    // observe-only target adjustment (no effect yet)
    CASE VO_Zone_Policy_Class[L_i] OF
        0: // comfort
            VO_Zone_Target_Adjustment[L_i] := 0.0;
            VO_Zone_Priority_Bias[L_i] := 1.0;

        1: // mild eco
            VO_Zone_Target_Adjustment[L_i] := -1.0;
            VO_Zone_Priority_Bias[L_i] := 0.8;

        2: // deep eco
            VO_Zone_Target_Adjustment[L_i] := -3.0;
            VO_Zone_Priority_Bias[L_i] := 0.5;

        3: // guest preheat
            VO_Zone_Target_Adjustment[L_i] := 0.0;
            VO_Zone_Priority_Bias[L_i] := 1.5;

        4: // permanent-use mild eco
            VO_Zone_Target_Adjustment[L_i] := -0.5;
            VO_Zone_Priority_Bias[L_i] := 0.9;

    END_CASE;

END_FOR;
          
END_FUNCTION_BLOCK

FUNCTION_BLOCK FB_Persist_Builder
  VAR_IN_OUT
    VIO_PersistStruct : ST_Persist;
  END_VAR

            // === BUILD STRUCT FROM STATE ===
// === NVRAM SNAPSHOT VIA STRUCT ADAPTER ===
VIO_PersistStruct.System_Mode := GVL_STATE.G_System_Mode;

VIO_PersistStruct.Safety_Gas_Latched := GVL_STATE.G_Safety_Gas_Latched;
VIO_PersistStruct.Safety_Smoke_Latched := GVL_STATE.G_Safety_Smoke_Latched;
VIO_PersistStruct.Safety_Leak_Latched := GVL_STATE.G_Safety_Leak_Latched;

VIO_PersistStruct.DHW_Heating_Pump := GVL_STATE.G_DHW_Heating_Pump;
VIO_PersistStruct.Valid := TRUE;

// mirror to legacy persistent variables
GVL_PERSISTENT.P_System_Mode := VIO_PersistStruct.System_Mode;

GVL_PERSISTENT.P_Safety_Gas_Latched := VIO_PersistStruct.Safety_Gas_Latched;
GVL_PERSISTENT.P_Safety_Smoke_Latched := VIO_PersistStruct.Safety_Smoke_Latched;
GVL_PERSISTENT.P_Safety_Leak_Latched := VIO_PersistStruct.Safety_Leak_Latched;

GVL_PERSISTENT.P_DHW_Heating_Active := VIO_PersistStruct.DHW_Heating_Pump;
GVL_PERSISTENT.P_Valid := VIO_PersistStruct.Valid;
          
END_FUNCTION_BLOCK

FUNCTION_BLOCK FB_Valve_Test_Manager
  VAR_INPUT
    VI_System_Time_MS : UDINT;
    VI_IsActivePLC : BOOL;
  END_VAR
  VAR_OUTPUT
    VO_Test_Active : BOOL;
    VO_Current_Valve : INT;
    VO_Valve_Cmd : ARRAY[1..GVL_CONSTANTS.C_MAX_MANIFOLDS] OF BOOL;
    VO_Test_Results : ARRAY[1..GVL_CONSTANTS.C_MAX_MANIFOLDS] OF BOOL;
    VO_Status_Msg : STRING(200);
  END_VAR
  VAR_IN_OUT
    VI_Valve_Currents : ARRAY[1..GVL_CONSTANTS.C_MAX_MANIFOLDS] OF REAL;
    VI_Valve_End_Switches : ARRAY[1..GVL_CONSTANTS.C_MAX_MANIFOLDS] OF BOOL;
    VI_Config : ARRAY[1..GVL_CONSTANTS.C_MAX_MANIFOLDS] OF ST_Valve_Test_Config;
  END_VAR
  VAR
    L_State : INT;
    L_Current_Valve : INT := 1;
    L_Test_Start_Time : UDINT;
    L_Last_Test_Time : ARRAY[1..GVL_CONSTANTS.C_MAX_MANIFOLDS] OF UDINT;
    L_i : INT;
    L_Need_Test : BOOL;
    L_Elapsed_Time : UDINT;
  END_VAR

            IF NOT VI_IsActivePLC THEN RETURN; END_IF;

CASE L_State OF
    0: // Ожидание
        VO_Test_Active := FALSE;
        L_Need_Test := FALSE;
        
        // Поиск клапана, которому нужен тест (раз в неделю)
        FOR L_i := 1 TO GVL_CONSTANTS.C_MAX_MANIFOLDS DO
            IF VI_Config[L_i].enabled AND ((VI_System_Time_MS - L_Last_Test_Time[L_i]) > (VI_Config[L_i].test_interval_days * 86400000)) THEN
                L_Current_Valve := L_i;
                L_Need_Test := TRUE;
                EXIT;
            END_IF;
        END_FOR;
        
        IF L_Need_Test THEN
            L_State := 1;
            L_Test_Start_Time := VI_System_Time_MS;
            VO_Test_Active := TRUE;
            VO_Current_Valve := L_Current_Valve;
            VO_Valve_Cmd[L_Current_Valve] := TRUE; // Открываем
            VO_Status_Msg := CONCAT('ТЕСТ КЛАПАНА ', INT_TO_STRING(L_Current_Valve));
            VO_Test_Results[L_Current_Valve] := TRUE; // Сброс результата
        END_IF;
        
    1: // Тестирование (ожидание открытия)
        L_Elapsed_Time := (VI_System_Time_MS - L_Test_Start_Time);
        
        IF VI_Valve_End_Switches[L_Current_Valve] THEN
            // Концевик сработал до истечения таймаута
            // Проверка тока
            IF ABS(VI_Valve_Currents[L_Current_Valve] - VI_Config[L_Current_Valve].Nominal_Current) > (VI_Config[L_Current_Valve].Nominal_Current * 0.2) THEN
                VO_Test_Results[L_Current_Valve] := FALSE; // Ошибка по току
            END_IF;
            
            GVL_Retain.G_Valve_Test_Results[L_Current_Valve] := VO_Test_Results[L_Current_Valve];
            
            VO_Valve_Cmd[L_Current_Valve] := FALSE; // Закрываем
            L_Test_Start_Time := VI_System_Time_MS; // Перезапускаем таймер для проверки закрытия
            L_State := 2;
        ELSIF L_Elapsed_Time > TO_UDINT(VI_Config[L_Current_Valve].nominal_close_time_sec * 1000.0) THEN
            // Таймаут открытия (заклинивание)
            VO_Test_Results[L_Current_Valve] := FALSE; 
            GVL_Retain.G_Valve_Test_Results[L_Current_Valve] := FALSE;
            VO_Status_Msg := CONCAT('ОШИБКА: ЗАКЛИНИВАНИЕ КЛАПАНА ', INT_TO_STRING(L_Current_Valve));
            
            VO_Valve_Cmd[L_Current_Valve] := FALSE; // Закрываем
            L_Test_Start_Time := VI_System_Time_MS; // Перезапускаем таймер
            L_State := 2;
        END_IF;
        
    2: // Ожидание закрытия
        L_Elapsed_Time := (VI_System_Time_MS - L_Test_Start_Time);
        
        IF NOT VI_Valve_End_Switches[L_Current_Valve] THEN
            // Концевик разомкнулся (клапан закрыт)
            L_Last_Test_Time[L_Current_Valve] := VI_System_Time_MS;
            L_State := 0;
            IF VO_Test_Results[L_Current_Valve] THEN
                VO_Status_Msg := 'ТЕСТ ЗАВЕРШЕН УСПЕШНО';
            END_IF;
        ELSIF L_Elapsed_Time > TO_UDINT(VI_Config[L_Current_Valve].nominal_close_time_sec * 1000.0) THEN
            // Таймаут закрытия (заклинивание)
            VO_Test_Results[L_Current_Valve] := FALSE; 
            GVL_Retain.G_Valve_Test_Results[L_Current_Valve] := FALSE;
            VO_Status_Msg := CONCAT('ОШИБКА: НЕ ЗАКРЫЛСЯ КЛАПАН ', INT_TO_STRING(L_Current_Valve));
            
            L_Last_Test_Time[L_Current_Valve] := VI_System_Time_MS;
            L_State := 0;
        END_IF;
END_CASE;
          
END_FUNCTION_BLOCK

FUNCTION_BLOCK FB_Water_Leakage_Manager
  VAR_INPUT
    VI_System_Time_MS : UDINT;
    VI_IsActivePLC : BOOL;
    VI_Config : ST_Flood_Global_Config;
  END_VAR
  VAR_OUTPUT
    VO_Status_Msg : STRING(200);
    VO_Leak_Detected : BOOL;
    VO_Leak_Warning_Level : BOOL;
  END_VAR
  VAR_IN_OUT
    VI_Sensors : ARRAY[1..GVL_CONSTANTS.C_MAX_FLOOD_SENSORS] OF BOOL;
  END_VAR
  VAR
    L_i : INT;
    L_Sensor_Timers : ARRAY[1..GVL_CONSTANTS.C_MAX_FLOOD_SENSORS] OF FB_System_Timer;
    L_Any_Leak : BOOL;
    L_Any_Warning : BOOL;
  END_VAR

            IF NOT VI_IsActivePLC THEN RETURN; END_IF;

L_Any_Leak := FALSE;
L_Any_Warning := FALSE;

FOR L_i := 1 TO GVL_CONSTANTS.C_MAX_FLOOD_SENSORS DO
    L_Sensor_Timers[L_i](
        IN := VI_Sensors[L_i],
        PT := TO_TIME(VI_Config.min_duration_ms + VI_Config.warning_duration_ms),
        VI_System_Time_MS := VI_System_Time_MS
    );

    IF L_Sensor_Timers[L_i].ET >= TO_TIME(VI_Config.min_duration_ms) THEN
        L_Any_Warning := TRUE;

        IF L_Sensor_Timers[L_i].Q THEN
            L_Any_Leak := TRUE;
        END_IF;
    END_IF;
END_FOR;

// Health signals
VO_Leak_Detected := L_Any_Leak;
VO_Leak_Warning_Level := L_Any_Warning;

// Status
IF L_Any_Leak THEN
    VO_Status_Msg := 'АВАРИЯ: ПРОТЕЧКА ВОДЫ.';
ELSIF L_Any_Warning THEN
    VO_Status_Msg := 'ПРЕДУПРЕЖДЕНИЕ: ОБНАРУЖЕНА ВОДА.';
ELSE
    VO_Status_Msg := 'Система контроля протечек в норме';
END_IF;
// >>> BULK_SYNC_ANCHOR: FB_Water_Leakage_Manager <<<
          
END_FUNCTION_BLOCK

FUNCTION_BLOCK FB_Scenario_Transition_Controller
  VAR_INPUT
    VI_System_Time : UDINT;
    VI_Start_Time : UDINT;
    VI_Duration : UDINT;
    VI_Start_Value : REAL;
    VI_End_Value : REAL;
  END_VAR
  VAR_OUTPUT
    VO_Current_Value : REAL;
    VO_Transition_Done : BOOL;
  END_VAR
  VAR
    L_Elapsed : UDINT;
    L_Progress : REAL;
  END_VAR

            L_Elapsed := (SEL(VI_System_Time >= VI_Start_Time, VI_System_Time - VI_Start_Time, (4294967295 - VI_Start_Time) + VI_System_Time + 1));

IF L_Elapsed >= VI_Duration OR VI_Duration = 0 THEN
    VO_Current_Value := VI_End_Value;
    VO_Transition_Done := TRUE;
ELSE
    L_Progress := UDINT_TO_REAL(L_Elapsed) / UDINT_TO_REAL(VI_Duration);
    VO_Current_Value := VI_Start_Value + (VI_End_Value - VI_Start_Value) * L_Progress;
    VO_Transition_Done := FALSE;
END_IF;
          
END_FUNCTION_BLOCK

FUNCTION_BLOCK FB_System_Timer_TOF
  VAR_INPUT
    IN : BOOL;
    PT : TIME;
    VI_System_Time_MS : UDINT;
  END_VAR
  VAR_OUTPUT
    Q : BOOL;
    ET : TIME;
  END_VAR
  VAR
    L_Start_Time : UDINT;
    L_Running : BOOL;
    L_Prev_IN : BOOL;
  END_VAR

            // ==============================================================================
// Блок таймера задержки выключения (System Timer TOF)
// Назначение:
// - Замена стандартного TOF для обеспечения точной выдержки времени,
//   независимой от времени цикла ПЛК, с использованием единого системного времени.
// ==============================================================================



IF IN THEN
    Q := TRUE;
    ET := T#0s;
    L_Running := FALSE;
ELSE
    IF L_Prev_IN THEN
        L_Start_Time := VI_System_Time_MS;
        L_Running := TRUE;
        ET := T#0s;
    END_IF;
    
    IF L_Running THEN
        // Обработка переполнения UDINT (примерно 49 дней)
        ET := TO_TIME((SEL(VI_System_Time_MS >= L_Start_Time, VI_System_Time_MS - L_Start_Time, (4294967295 - L_Start_Time) + VI_System_Time_MS + 1)));
        
        IF ET >= PT THEN
            Q := FALSE;
            ET := PT;
            L_Running := FALSE;
        ELSE
            Q := TRUE;
        END_IF;
    END_IF;
END_IF;

L_Prev_IN := IN;
          
END_FUNCTION_BLOCK

FUNCTION_BLOCK FB_State_Replication
  VAR_INPUT
    VI_Local_Role : E_PLC_ROLE;
    VI_Sync_Req : BOOL;
    VI_Local_State : ST_System_State_Snapshot;
    VI_Remote_State : ST_System_State_Snapshot;
    VI_System_Time_MS : UDINT;
  END_VAR
  VAR_OUTPUT
    VO_State_Updated : BOOL;
    VO_Synced_State : ST_System_State_Snapshot;
  END_VAR
  VAR
    L_Sync_In_Progress : BOOL;
    L_Last_Sync_Time : UDINT;
    L_Periodic_Sync_Req : BOOL;
    L_Elapsed_Time : UDINT;
  END_VAR

            // Периодическая синхронизация (каждые 5 секунд)
L_Elapsed_Time := (SEL(VI_System_Time_MS >= L_Last_Sync_Time, VI_System_Time_MS - L_Last_Sync_Time, (4294967295 - L_Last_Sync_Time) + VI_System_Time_MS + 1));

IF L_Elapsed_Time > 5000 THEN
    L_Periodic_Sync_Req := TRUE;
    L_Last_Sync_Time := VI_System_Time_MS;
ELSE
    L_Periodic_Sync_Req := FALSE;
END_IF;

// State Replication Logic
// Синхронизация состояния между ПЛК (ТЗ 8.2)
IF (VI_Sync_Req OR L_Periodic_Sync_Req) AND NOT L_Sync_In_Progress THEN
    L_Sync_In_Progress := TRUE;
    
    // Разрешение конфликтов на основе версии состояния
    IF VI_Remote_State.Version > VI_Local_State.Version THEN
        VO_Synced_State := VI_Remote_State;
        VO_State_Updated := TRUE;
    ELSIF VI_Remote_State.Version = VI_Local_State.Version THEN
        // Если версии равны, приоритет у ведущего ПЛК
        IF VI_Local_Role = E_PLC_ROLE.ROLE_STANDBY THEN
            VO_Synced_State := VI_Remote_State;
            VO_State_Updated := TRUE;
        ELSE
            VO_Synced_State := VI_Local_State;
            VO_State_Updated := FALSE;
        END_IF;
    ELSE
        VO_Synced_State := VI_Local_State;
        VO_State_Updated := FALSE;
    END_IF;
ELSIF NOT (VI_Sync_Req OR L_Periodic_Sync_Req) THEN
    L_Sync_In_Progress := FALSE;
    VO_State_Updated := FALSE;
    VO_Synced_State := VI_Local_State;
END_IF;
          
END_FUNCTION_BLOCK

FUNCTION_BLOCK FB_Gateway_Interface
  VAR_INPUT
    VI_System_Time_MS : UDINT;
    VI_Local_PLC_Role : E_PLC_ROLE;
    VI_Incoming_Command : ST_Gateway_Command;
    VI_Command_Received : BOOL;
    VI_Outdoor_Temp : REAL;
    VI_Security_Armed : BOOL;
    VI_Flood_Alarm_Active : BOOL;
    VI_Gas_Alarm_Active : BOOL;
    VI_Fire_Alarm_Active : BOOL;
    VI_Methane_Concentration : REAL;
    VI_Active_Scenario : E_SCENARIO_TYPE;
    VI_Send_2FA_Req : BOOL;
    VI_2FA_Code : STRING(6);
  END_VAR
  VAR_OUTPUT
    VO_Modbus_Registers : ARRAY[0..GVL_CONSTANTS.C_MAX_MODBUS_REGISTERS-1] OF WORD;
    VO_Lighting_Override : ARRAY[1..32] OF BYTE;
    VO_Blinds_Override : ARRAY[1..GVL_CONSTANTS.C_MAX_BLINDS] OF BYTE;
    VO_Socket_Override : ARRAY[1..GVL_CONSTANTS.C_MAX_SOCKETS] OF BOOL;
    VO_Arm_Req : BOOL;
    VO_Disarm_Req : BOOL;
    VO_PIN_Code : STRING(4);
    VO_RFID_Tag : STRING(20);
    VO_2FA_Code_In : STRING(6);
    VO_Data_Ready : BOOL;
    VO_HMI_Status_Message : STRING(200);
    VO_Telegram_Msg : STRING(200);
    VO_Send_Telegram : BOOL;
    VO_Set_Scenario_Req : BOOL;
    VO_Target_Scenario : E_SCENARIO_TYPE;
    VO_Set_Temp_Req : BOOL;
    VO_Target_Zone : INT;
    VO_Target_Temp : REAL;
    VO_Set_Vent_Req : BOOL;
    VO_Target_Vent_Speed : BYTE;
    VO_Reset_Errors_Req : BOOL;
    VO_Set_Config_Req : BOOL;
    VO_Sync_Time_Req : BOOL;
    VO_New_Time_MS : UDINT;
  END_VAR
  VAR_IN_OUT
    VI_FloorHeating_Temps : ARRAY[1..8] OF REAL;
    VI_Room_Temps : ARRAY[1..16] OF REAL;
    VI_Zone_Valve_States : ARRAY[1..8] OF BOOL;
    VI_Manifold_Pressures : ARRAY[1..GVL_CONSTANTS.C_MAX_MANIFOLDS] OF REAL;
    VI_Manifold_Pump_States : ARRAY[1..GVL_CONSTANTS.C_MAX_MANIFOLDS] OF BOOL;
    VI_Lighting_Base_Levels : ARRAY[1..32] OF BYTE;
    VI_Socket_States : ARRAY[1..GVL_CONSTANTS.C_MAX_SOCKETS] OF BOOL;
    VI_Blinds_Positions : ARRAY[1..GVL_CONSTANTS.C_MAX_BLINDS] OF BYTE;
    VI_Allowed_IPs : ARRAY[1..GVL_CONSTANTS.C_MAX_ALLOWED_IPS] OF STRING(15);
  END_VAR
  VAR
    L_last_update_time : UDINT;
    L_i : INT;
    L_j : INT;
    L_idx : INT;
    L_tmp_word : WORD;
    L_Code_UDINT : UDINT;
    L_Prev_Fire : BOOL;
    L_Prev_Gas : BOOL;
    L_Prev_Flood : BOOL;
    L_Prev_Security : BOOL;
    L_Deduplicator : FB_Command_Deduplication;
    L_CRC_Calc : FB_CRC32_Calculator;
    L_Calculated_CRC : DWORD;
    L_Command_Size : UDINT;
    L_IP_Allowed : BOOL;
    L_Process_Command : ST_Gateway_Command;
    L_Has_Command_To_Process : BOOL;
  END_VAR
  VAR RETAIN
    L_Command_Buffer : ARRAY[1..GVL_CONSTANTS.C_MAX_GATEWAY_COMMANDS] OF ST_Gateway_Command;
    L_Buffer_Head : INT := 1;
    L_Buffer_Tail : INT := 1;
    L_Buffer_Count : INT := 0;
  END_VAR

            // Отправка уведомлений в Telegram (ТЗ 10.2)
VO_Send_Telegram := FALSE;
IF VI_Fire_Alarm_Active AND NOT L_Prev_Fire THEN
    VO_Telegram_Msg := 'ВНИМАНИЕ! ПОЖАРНАЯ ТРЕВОГА!';
    VO_Send_Telegram := TRUE;
END_IF;
IF VI_Gas_Alarm_Active AND NOT L_Prev_Gas THEN
    VO_Telegram_Msg := 'ВНИМАНИЕ! УТЕЧКА ГАЗА!';
    VO_Send_Telegram := TRUE;
END_IF;
IF VI_Flood_Alarm_Active AND NOT L_Prev_Flood THEN
    VO_Telegram_Msg := 'ВНИМАНИЕ! ПРОТЕЧКА ВОДЫ!';
    VO_Send_Telegram := TRUE;
END_IF;
IF VI_Security_Armed AND NOT L_Prev_Security THEN
    VO_Telegram_Msg := 'ОХРАНА ВКЛЮЧЕНА';
    VO_Send_Telegram := TRUE;
ELSIF NOT VI_Security_Armed AND L_Prev_Security THEN
    VO_Telegram_Msg := 'ОХРАНА ОТКЛЮЧЕНА';
    VO_Send_Telegram := TRUE;
END_IF;

L_Prev_Fire := VI_Fire_Alarm_Active;
L_Prev_Gas := VI_Gas_Alarm_Active;
L_Prev_Flood := VI_Flood_Alarm_Active;
L_Prev_Security := VI_Security_Armed;

// Обновление данных Modbus (раз в 1 сек)
IF (VI_System_Time_MS - L_last_update_time) >= GVL_CONSTANTS.C_MS_IN_SECOND THEN
    L_last_update_time := VI_System_Time_MS;
    
    // 0: Статус ПЛК и Аварии
    L_tmp_word := 0;
    IF VI_Local_PLC_Role = E_PLC_ROLE.ROLE_ACTIVE THEN L_tmp_word := L_tmp_word OR 1; END_IF;
    IF VI_Security_Armed THEN L_tmp_word := L_tmp_word OR 2; END_IF;
    IF VI_Flood_Alarm_Active THEN L_tmp_word := L_tmp_word OR 4; END_IF;
    IF VI_Gas_Alarm_Active THEN L_tmp_word := L_tmp_word OR 8; END_IF;
    IF VI_Fire_Alarm_Active THEN L_tmp_word := L_tmp_word OR 16; END_IF;
    VO_Modbus_Registers[0] := L_tmp_word;

    // 1-16: Температуры пола (x10)
    FOR L_i := 1 TO 8 DO
        VO_Modbus_Registers[L_i] := TO_WORD(TO_INT(VI_FloorHeating_Temps[L_i] * 10.0));
    END_FOR;

    // 17-310102: Температуры помещений (x10)
    FOR L_i := 1 TO 16 DO
        VO_Modbus_Registers[16 + L_i] := TO_WORD(TO_INT(VI_Room_Temps[L_i] * 10.0));
    END_FOR;

    // 310103: Состояние клапанов зон (битовая маска 1-16)
    L_tmp_word := 0;
    FOR L_i := 1 TO 8 DO
        IF VI_Zone_Valve_States[L_i] THEN
            L_tmp_word := L_tmp_word OR SHL(TO_WORD(1), L_i - 1);
        END_IF;
    END_FOR;
    VO_Modbus_Registers[33] := L_tmp_word;

    // 34-38: Давление в коллекторах (x100)
    FOR L_i := 1 TO GVL_CONSTANTS.C_MAX_MANIFOLDS DO
        VO_Modbus_Registers[33 + L_i] := TO_WORD(TO_INT(VI_Manifold_Pressures[L_i] * 100.0));
    END_FOR;

    // 40-55: Базовое освещение
    FOR L_i := 1 TO 32 DO
        VO_Modbus_Registers[39 + L_i] := TO_WORD(VI_Lighting_Base_Levels[L_i]);
    END_FOR;

    // 60-79: Положение штор (20 шт)
    FOR L_i := 1 TO GVL_CONSTANTS.C_MAX_BLINDS DO
        VO_Modbus_Registers[59 + L_i] := TO_WORD(VI_Blinds_Positions[L_i]);
    END_FOR;

    // 80-82: Розетки (битовая маска, 36 розеток -> 3 WORD)
    FOR L_i := 0 TO (GVL_CONSTANTS.C_MAX_SOCKETS - 1) / 16 DO
        L_tmp_word := 0;
        FOR L_j := 1 TO 16 DO
            L_idx := (L_i * 16) + L_j;
            IF L_idx <= GVL_CONSTANTS.C_MAX_SOCKETS THEN
                IF VI_Socket_States[L_idx] THEN
                    L_tmp_word := L_tmp_word OR SHL(TO_WORD(1), L_j - 1);
                END_IF;
            END_IF;
        END_FOR;
        VO_Modbus_Registers[79 + L_i] := L_tmp_word;
    END_FOR;

    // 100-102: 2FA Request and Code
    VO_Modbus_Registers[100] := SEL(VI_Send_2FA_Req, 0, 1);
    IF VI_Send_2FA_Req THEN
        L_Code_UDINT := STRING_TO_UDINT(VI_2FA_Code);
        VO_Modbus_Registers[101] := TO_WORD(L_Code_UDINT AND 16#FFFF);
        VO_Modbus_Registers[102] := TO_WORD(SHR(L_Code_UDINT, 16));
    ELSE
        VO_Modbus_Registers[101] := 0;
        VO_Modbus_Registers[102] := 0;
    END_IF;

    VO_Data_Ready := TRUE;
END_IF;

// Обработка входящих команд
VO_Arm_Req := FALSE;
VO_Disarm_Req := FALSE;
VO_Set_Scenario_Req := FALSE;
VO_Set_Temp_Req := FALSE;
VO_Set_Vent_Req := FALSE;
VO_Reset_Errors_Req := FALSE;
VO_Set_Config_Req := FALSE;
VO_Sync_Time_Req := FALSE;
L_Has_Command_To_Process := FALSE;

// 1. Прием команды и буферизация
IF VI_Command_Received THEN
    IF VI_Local_PLC_Role = E_PLC_ROLE.ROLE_ACTIVE THEN
        // Если активен, обрабатываем сразу
        L_Process_Command := VI_Incoming_Command;
        L_Has_Command_To_Process := TRUE;
    ELSE
        // Если резервный, добавляем в буфер
        IF L_Buffer_Count < GVL_CONSTANTS.C_MAX_GATEWAY_COMMANDS THEN
            L_Command_Buffer[L_Buffer_Head] := VI_Incoming_Command;
            L_Buffer_Head := L_Buffer_Head + 1;
            IF L_Buffer_Head > GVL_CONSTANTS.C_MAX_GATEWAY_COMMANDS THEN L_Buffer_Head := 1; END_IF;
            L_Buffer_Count := L_Buffer_Count + 1;
        END_IF;
    END_IF;
END_IF;

// 2. Извлечение из буфера при переходе в активный режим
IF NOT L_Has_Command_To_Process AND (VI_Local_PLC_Role = E_PLC_ROLE.ROLE_ACTIVE) AND (L_Buffer_Count > 0) THEN
    L_Process_Command := L_Command_Buffer[L_Buffer_Tail];
    L_Buffer_Tail := L_Buffer_Tail + 1;
    IF L_Buffer_Tail > GVL_CONSTANTS.C_MAX_GATEWAY_COMMANDS THEN L_Buffer_Tail := 1; END_IF;
    L_Buffer_Count := L_Buffer_Count - 1;
    L_Has_Command_To_Process := TRUE;
END_IF;

// 3. Обработка команды
IF L_Has_Command_To_Process THEN
    // Проверка IP-адреса источника
    L_IP_Allowed := FALSE;
    IF L_Process_Command.source_ip = '' THEN
        L_IP_Allowed := TRUE; // Если IP не передан, пропускаем (для обратной совместимости или локальных вызовов)
    ELSE
        FOR L_i := 1 TO GVL_CONSTANTS.C_MAX_ALLOWED_IPS DO
            IF VI_Allowed_IPs[L_i] = L_Process_Command.source_ip THEN
                L_IP_Allowed := TRUE;
                EXIT;
            END_IF;
        END_FOR;
    END_IF;
    
    IF NOT L_IP_Allowed THEN
        VO_HMI_Status_Message := 'Gateway: Ошибка безопасности (Неизвестный IP)';
        RETURN;
    END_IF;

    // Проверка целостности данных (CRC32)
    // Размер данных для расчета CRC: размер структуры минус размер самого поля crc32
    L_Command_Size := SIZEOF(L_Process_Command) - SIZEOF(L_Process_Command.crc32);
    L_Calculated_CRC := L_CRC_Calc.Calculate();
    
    IF L_Calculated_CRC = L_Process_Command.crc32 THEN
        L_Deduplicator(
            VI_Command_ID := L_Process_Command.command_id,
            VI_Command_Type := L_Process_Command.command_type,
            VI_Command_Value := L_Process_Command.target_value,
            VI_System_Time_MS := VI_System_Time_MS
        );
        
        IF L_Deduplicator.VO_Is_New_Command THEN
            CASE L_Process_Command.command_type OF
        E_Gateway_Command_Type.CMD_SET_SCENARIO: // Управление сценариями
            VO_Set_Scenario_Req := TRUE;
            VO_Target_Scenario := L_Process_Command.target_scenario;
            VO_HMI_Status_Message := 'Gateway: Сценарий изменен';
        E_Gateway_Command_Type.CMD_SET_LIGHT: // Управление освещением
            IF (L_Process_Command.target_zone >= 1) AND (L_Process_Command.target_zone <= 32) THEN
                VO_Lighting_Override[L_Process_Command.target_zone] := TO_BYTE(L_Process_Command.target_value);
                VO_HMI_Status_Message := 'Gateway: Команда освещения принята';
            END_IF;
        E_Gateway_Command_Type.CMD_SET_BLINDS: // Управление шторами
            IF (L_Process_Command.target_zone >= 1) AND (L_Process_Command.target_zone <= GVL_CONSTANTS.C_MAX_BLINDS) THEN
                VO_Blinds_Override[L_Process_Command.target_zone] := TO_BYTE(L_Process_Command.target_value);
                VO_HMI_Status_Message := 'Gateway: Команда штор принята';
            END_IF;
        E_Gateway_Command_Type.CMD_SET_SOCKET: // Розетки
            IF (L_Process_Command.target_zone >= 1) AND (L_Process_Command.target_zone <= GVL_CONSTANTS.C_MAX_SOCKETS) THEN
                VO_Socket_Override[L_Process_Command.target_zone] := L_Process_Command.target_on_off;
                VO_HMI_Status_Message := 'Gateway: Команда розетки принята';
            END_IF;
        E_Gateway_Command_Type.CMD_SET_SECURITY: // Охрана
            IF L_Process_Command.target_armed THEN
                VO_Arm_Req := TRUE;
            ELSE
                VO_Disarm_Req := TRUE;
            END_IF;
            VO_PIN_Code := L_Process_Command.target_pin;
            VO_2FA_Code_In := L_Process_Command.target_2fa_code;
            VO_HMI_Status_Message := 'Gateway: Запрос охраны принят';
        E_Gateway_Command_Type.CMD_SET_TEMP: // Управление температурой
            IF (L_Process_Command.target_zone >= 1) AND (L_Process_Command.target_zone <= 32) THEN
                VO_Set_Temp_Req := TRUE;
                VO_Target_Zone := L_Process_Command.target_zone;
                VO_Target_Temp := L_Process_Command.target_value;
                VO_HMI_Status_Message := 'Gateway: Уставка температуры изменена';
            END_IF;
        E_Gateway_Command_Type.CMD_SET_VENT: // Управление вентиляцией
            // Пример: изменение скорости притока
            VO_Set_Vent_Req := TRUE;
            VO_Target_Vent_Speed := TO_BYTE(L_Process_Command.target_value);
            VO_HMI_Status_Message := 'Gateway: Уставка вентиляции изменена';
        E_Gateway_Command_Type.CMD_TELEGRAM_MSG: // Отправка сообщения в Telegram
            VO_Telegram_Msg := L_Process_Command.telegram_msg;
            VO_Send_Telegram := TRUE;
            VO_HMI_Status_Message := 'Gateway: Сообщение Telegram отправлено';

        E_Gateway_Command_Type.CMD_SYNC_TIME: // Синхронизация времени
            VO_Sync_Time_Req := TRUE;
            VO_New_Time_MS := TO_UDINT(L_Process_Command.target_value);
            VO_HMI_Status_Message := 'Gateway: Время синхронизировано';

        E_Gateway_Command_Type.CMD_RESET_ERRORS: // Квитирование / сброс ошибок
            VO_Reset_Errors_Req := TRUE;
            VO_HMI_Status_Message := 'Gateway: Запрос на сброс ошибок принят';

        E_Gateway_Command_Type.CMD_SET_CONFIG: // Применение конфигурации
            VO_Set_Config_Req := TRUE;
            VO_HMI_Status_Message := 'Gateway: Запрос на применение конфигурации принят';
        END_CASE;
    END_IF;
ELSE
    VO_HMI_Status_Message := 'Gateway: Ошибка CRC команды';
END_IF;
END_IF;
// >>> BULK_SYNC_ANCHOR: FB_Gateway_Interface <<<
          
END_FUNCTION_BLOCK

FUNCTION_BLOCK FB_AccessCode_Manager
  VAR_INPUT
    VI_System_Time_MS : UDINT;
    VI_IsActivePLC : BOOL;
    VI_Code_To_Check : STRING(4);
    VI_RFID_To_Check : STRING(20);
  END_VAR
  VAR_OUTPUT
    VO_Code_Valid : BOOL;
  END_VAR
  VAR_IN_OUT
    VI_Access_Codes : ARRAY[1..GVL_CONSTANTS.C_MAX_ACCESS_CODES] OF DWORD;
    VI_RFID_Tags : ARRAY[1..GVL_CONSTANTS.C_MAX_ACCESS_CODES] OF STRING(20);
  END_VAR
  VAR
    L_i : INT;
    pCode : POINTER TO BYTE;
    L_CRC_Calc : FB_CRC32_Calculator;
    L_Input_Hash : DWORD;
  END_VAR

            VO_Code_Valid := FALSE;

// Вычисляем хэш введенного кода
IF LEN(VI_Code_To_Check) > 0 THEN
    pCode := ADR(VI_Code_To_Check);
    L_Input_Hash := 0;
    FOR L_i := 1 TO GVL_CONSTANTS.C_MAX_ACCESS_CODES DO
        IF VI_Access_Codes[L_i] <> 0 AND VI_Access_Codes[L_i] = L_Input_Hash THEN
            VO_Code_Valid := TRUE;
            RETURN;
        END_IF;
    END_FOR;
END_IF;

// Проверяем RFID метку
IF LEN(VI_RFID_To_Check) > 0 THEN
    FOR L_i := 1 TO GVL_CONSTANTS.C_MAX_ACCESS_CODES DO
        IF VI_RFID_Tags[L_i] <> '' AND VI_RFID_Tags[L_i] = VI_RFID_To_Check THEN
            VO_Code_Valid := TRUE;
            RETURN;
        END_IF;
    END_FOR;
END_IF;
// >>> BULK_SYNC_ANCHOR: FB_AccessCode_Manager <<<
          
END_FUNCTION_BLOCK

FUNCTION_BLOCK FB_Presence_Manager
  VAR_INPUT
    VI_Motion_Sensors : ARRAY[1..32] OF BOOL;
    VI_System_Time_MS : UDINT;
  END_VAR
  VAR_OUTPUT
    VO_Any_Motion : BOOL;
    VO_Occupied : BOOL;
    VO_Auto_Away : BOOL;
    VO_Last_Motion_TS : UDINT;
  END_VAR
  VAR
    L_Last_Motion_TS : UDINT := 0;
    L_Initialized : BOOL := FALSE;
    L_Timeout_MS : UDINT := 900000;
    L_i : INT;
  END_VAR

            // detect any motion
VO_Any_Motion := FALSE;
FOR L_i := 1 TO 32 DO
    IF VI_Motion_Sensors[L_i] THEN
        VO_Any_Motion := TRUE;
    END_IF;
END_FOR;

// init protection (avoid instant AWAY at boot)
IF NOT L_Initialized THEN
    L_Last_Motion_TS := VI_System_Time_MS;
    L_Initialized := TRUE;
END_IF;

// fast return: any motion immediately updates timestamp
IF VO_Any_Motion THEN
    L_Last_Motion_TS := VI_System_Time_MS;
END_IF;

// hysteresis logic:
// stay OCCUPIED until timeout expires
IF (VI_System_Time_MS - L_Last_Motion_TS) < L_Timeout_MS THEN
    VO_Occupied := TRUE;
ELSE
    VO_Occupied := FALSE;
END_IF;

VO_Auto_Away := NOT VO_Occupied;
VO_Last_Motion_TS := L_Last_Motion_TS;
          
END_FUNCTION_BLOCK

FUNCTION_BLOCK FB_Astro_Timer
  VAR_INPUT
    VI_System_Time_MS : UDINT;
    VI_Latitude : REAL := 55.75;
    VI_Longitude : REAL := 37.61;
    VI_Timezone : REAL := 3.0;
    VI_Day_Of_Year : UINT;
  END_VAR
  VAR_OUTPUT
    VO_Sunset_Time : TOD;
    VO_Sunrise_Time : TOD;
    VO_Is_Night : BOOL;
    VO_Current_TOD : TOD;
  END_VAR
  VAR
    L_Current_TOD : TOD;
    L_Pi : REAL := 3.14159265359;
    L_Rad : REAL := 3.14159265359 / 180.0;
    L_Deg : REAL := 180.0 / 3.14159265359;
    L_B : REAL;
    L_EoT : REAL;
    L_Declination : REAL;
    L_Cos_Omega : REAL;
    L_Omega : REAL;
    L_Sunrise_Local : REAL;
    L_Sunset_Local : REAL;
  END_VAR

            // >>> SYNC_TEST_MARKER_002 <<<


L_Current_TOD := GVL_STATUS.G_Current_TOD;
VO_Current_TOD := L_Current_TOD;

// Equation of Time (EoT) in minutes
L_B := 360.0 / 365.0 * TO_REAL(VI_Day_Of_Year - 81) * L_Rad;
L_EoT := 9.87 * SIN(2.0 * L_B) - 7.53 * COS(L_B) - 1.5 * SIN(L_B);

// Solar Declination in degrees
L_Declination := 23.45 * SIN(360.0 / 365.0 * TO_REAL(VI_Day_Of_Year + 284) * L_Rad);

// Hour angle
L_Cos_Omega := -TAN(VI_Latitude * L_Rad) * TAN(L_Declination * L_Rad);

IF L_Cos_Omega > 1.0 THEN
    L_Cos_Omega := 1.0; // Polar night
ELSIF L_Cos_Omega < -1.0 THEN
    L_Cos_Omega := -1.0; // Polar day
END_IF;

L_Omega := ACOS(L_Cos_Omega) * L_Deg;

// Sunrise and Sunset in local time (hours)
L_Sunrise_Local := 12.0 - (L_Omega / 15.0) - (L_EoT / 60.0) + (VI_Timezone * 15.0 - VI_Longitude) / 15.0;
L_Sunset_Local := 12.0 + (L_Omega / 15.0) - (L_EoT / 60.0) + (VI_Timezone * 15.0 - VI_Longitude) / 15.0;

// Handle bounds
IF L_Sunrise_Local < 0.0 THEN L_Sunrise_Local := L_Sunrise_Local + 24.0; END_IF;
IF L_Sunrise_Local >= 24.0 THEN L_Sunrise_Local := L_Sunrise_Local - 24.0; END_IF;
IF L_Sunset_Local < 0.0 THEN L_Sunset_Local := L_Sunset_Local + 24.0; END_IF;
IF L_Sunset_Local >= 24.0 THEN L_Sunset_Local := L_Sunset_Local - 24.0; END_IF;

// Конвертация в TOD
VO_Sunrise_Time := TO_TOD(TO_UDINT(L_Sunrise_Local * 3600000.0));
VO_Sunset_Time := TO_TOD(TO_UDINT(L_Sunset_Local * 3600000.0));

// ТЗ 15.2: Закат + 30 мин / Рассвет - 30 мин
VO_Is_Night := (L_Current_TOD > (VO_Sunset_Time + T#30m)) OR (L_Current_TOD < (VO_Sunrise_Time - T#30m));
// >>> SYNC_TEST_MARKER_FORCE <<<
// >>> BULK_SYNC_ANCHOR: FB_Astro_Timer <<<
          
END_FUNCTION_BLOCK

FUNCTION_BLOCK FB_FloorHeating_Freeze_Protection
  VAR_INPUT
    VI_Outdoor_Temp : REAL;
    VI_Threshold : REAL := 7.0;
  END_VAR
  VAR_OUTPUT
    VO_Freeze_Alert : BOOL;
    VO_Pump_Force_On : BOOL;
  END_VAR
  VAR_IN_OUT
    VI_Floor_Temps : ARRAY[1..GVL_CONSTANTS.C_MAX_HEATING_CIRCUITS] OF REAL;
  END_VAR
  VAR
    L_i : INT;
  END_VAR

            VO_Freeze_Alert := FALSE;
VO_Pump_Force_On := FALSE;

FOR L_i := 1 TO GVL_CONSTANTS.C_MAX_HEATING_CIRCUITS DO
    IF VI_Floor_Temps[L_i] < VI_Threshold THEN
        VO_Freeze_Alert := TRUE;
        VO_Pump_Force_On := TRUE;
        RETURN;
    END_IF;
END_FOR;

IF VI_Outdoor_Temp < -5.0 THEN
    VO_Pump_Force_On := TRUE;
END_IF;
          
END_FUNCTION_BLOCK

PROGRAM PRG_Policy

            // ============================================================
// SCENARIO POLICY OWNER
// ============================================================

// 1. Base priority resolution
IF GVL_STATE.G_System_Mode = E_System_Operating_Mode.MODE_SAFE_STOP THEN
    GVL_POLICY.G_Scenario_Intent := E_SCENARIO_TYPE.SCENARIO_NONE;
    GVL_POLICY.G_Scenario_Source := SRC_SAFETY;

ELSIF GVL_POLICY.G_Scenario_Request_Operator <> E_SCENARIO_TYPE.SCENARIO_NONE THEN
    GVL_POLICY.G_Scenario_Intent := GVL_POLICY.G_Scenario_Request_Operator;
    GVL_POLICY.G_Scenario_Source := SRC_OPERATOR;

ELSIF GVL_POLICY.G_Scenario_Request_Gateway <> E_SCENARIO_TYPE.SCENARIO_NONE THEN
    GVL_POLICY.G_Scenario_Intent := GVL_POLICY.G_Scenario_Request_Gateway;
    GVL_POLICY.G_Scenario_Source := SRC_GATEWAY;

ELSIF GVL_POLICY.G_Scenario_Request_Rule <> E_SCENARIO_TYPE.SCENARIO_NONE THEN
    GVL_POLICY.G_Scenario_Intent := GVL_POLICY.G_Scenario_Request_Rule;
    GVL_POLICY.G_Scenario_Source := SRC_RULE;

ELSE
    GVL_POLICY.G_Scenario_Intent := GVL_STATUS.G_Current_Scenario;
    GVL_POLICY.G_Scenario_Source := SRC_NONE;
END_IF;

// 2. Fail-safe clamp
CASE GVL_STATE.G_System_Mode OF
    E_System_Operating_Mode.MODE_SAFE_STOP:
        GVL_POLICY.G_Scenario_Intent := E_SCENARIO_TYPE.SCENARIO_NONE;
        GVL_POLICY.G_Scenario_Source := SRC_SAFETY;

    E_System_Operating_Mode.MODE_FREEZE_PROTECTION:
        GVL_POLICY.G_Scenario_Intent := E_SCENARIO_TYPE.SCENARIO_NONE;
        GVL_POLICY.G_Scenario_Source := SRC_POLICY;

    E_System_Operating_Mode.MODE_DEGRADED:
        CASE GVL_POLICY.G_Scenario_Intent OF
            E_SCENARIO_TYPE.SCENARIO_NONE,
            E_SCENARIO_TYPE.SCENARIO_PRESENCE,
            E_SCENARIO_TYPE.SCENARIO_AWAY,
            E_SCENARIO_TYPE.SCENARIO_SLEEP:
                ;
        ELSE
            GVL_POLICY.G_Scenario_Intent := E_SCENARIO_TYPE.SCENARIO_NONE;
            GVL_POLICY.G_Scenario_Source := SRC_POLICY;
        END_CASE;
END_CASE;

// 3. Context automation
IF GVL_STATE.G_System_Mode = E_System_Operating_Mode.MODE_NORMAL THEN
    IF GVL_ALARM.G_Security_Armed AND
       (GVL_POLICY.G_Scenario_Request_Operator = E_SCENARIO_TYPE.SCENARIO_NONE) AND
       (GVL_POLICY.G_Scenario_Request_Gateway = E_SCENARIO_TYPE.SCENARIO_NONE) AND
       (GVL_POLICY.G_Scenario_Request_Rule = E_SCENARIO_TYPE.SCENARIO_NONE) AND
       (GVL_POLICY.G_Scenario_Intent <> E_SCENARIO_TYPE.SCENARIO_AWAY) THEN
        GVL_POLICY.G_Scenario_Intent := E_SCENARIO_TYPE.SCENARIO_AWAY;
        GVL_POLICY.G_Scenario_Source := SRC_POLICY;
    END_IF;
END_IF;

// 4. Degraded adaptation
IF GVL_STATE.G_System_Mode = E_System_Operating_Mode.MODE_DEGRADED THEN
    IF (GVL_POLICY.G_Scenario_Request_Operator = E_SCENARIO_TYPE.SCENARIO_NONE) AND
       (GVL_POLICY.G_Scenario_Request_Gateway = E_SCENARIO_TYPE.SCENARIO_NONE) AND
       (GVL_POLICY.G_Scenario_Request_Rule = E_SCENARIO_TYPE.SCENARIO_NONE) THEN

        IF GVL_ALARM.G_Security_Armed THEN
            GVL_POLICY.G_Scenario_Intent := E_SCENARIO_TYPE.SCENARIO_AWAY;
            GVL_POLICY.G_Scenario_Source := SRC_POLICY;

        ELSIF GVL_POLICY.G_Scenario_Intent = E_SCENARIO_TYPE.SCENARIO_PRESENCE THEN
            GVL_POLICY.G_Scenario_Intent := E_SCENARIO_TYPE.SCENARIO_SLEEP;
            GVL_POLICY.G_Scenario_Source := SRC_POLICY;
        END_IF;
    END_IF;
END_IF;

// 5. Heating bridge
GVL_STATE.G_Preheat_Request := GVL_POLICY.G_Rule_Preheat_Request;
GVL_STATE.G_Freeze_Request :=
    (GVL_STATE.G_System_Mode = E_System_Operating_Mode.MODE_FREEZE_PROTECTION);
          
END_PROGRAM

PROGRAM PRG_PLC_B

            // Вызов основной программы
PRG_System();
// >>> BULK_SYNC_ANCHOR: PRG_PLC_B <<<
          
END_PROGRAM

PROGRAM PRG_Scenario_Test_Harness
  VAR
    L_i : INT;
    L_j : INT;
    L_circuit : INT;
    L_manifold : INT;
    L_base : INT;
    L_expected : INT;
    L_actual : INT;
    L_tmp : INT;
    L_Manifold_Calc : ARRAY[1..GVL_CONSTANTS.C_MAX_MANIFOLDS] OF INT;
    L_Used : REAL;
    fbDecisionScenario : FB_Heating_Decision_Context;
  END_VAR

            // === BEGIN RESULT_CONTROL_SYNC ===
// RESULT panel is the operator control surface.
GVL_TEST_PANEL.G_Enable := GVL_TEST_PANEL_RESULT.G_Enable;
GVL_TEST_PANEL.G_Scenario_ID := GVL_TEST_PANEL_RESULT.G_Scenario_ID;
GVL_TEST_PANEL.G_Scenario_Run := GVL_TEST_PANEL_RESULT.G_Scenario_Run;
// === END RESULT_CONTROL_SYNC ===

IF NOT GVL_TEST_PANEL.G_Enable THEN
    RETURN;
END_IF;

// === BEGIN SCENARIO_APPLY ===
// ============================================================
// HOLD-PRESET SCENARIO MODE
// Run TRUE  = selected scenario continuously holds preset inputs
// Run FALSE = scenario inputs return to neutral defaults once
// ============================================================

IF GVL_TEST_PANEL.G_Scenario_Run THEN
    GVL_TEST_PANEL.G_Selected_Circuit := 1;
    GVL_TEST_PANEL.G_Input_Policy_Bias := 0;
    GVL_TEST_PANEL.G_Input_Guest_Preheat_Request := FALSE;
    GVL_TEST_PANEL.G_Input_Guest_Preheat_Enabled := TRUE;
    GVL_TEST_PANEL.G_Input_Guest_Preheat_Boost := 2;
    GVL_TEST_PANEL.G_Input_Max_Thermal_Budget := 2.0;
    GVL_TEST_PANEL.G_Input_Block_Heating := FALSE;
    GVL_TEST_PANEL.G_Input_Safety_Stop := FALSE;

    FOR L_i := 1 TO GVL_CONSTANTS.C_MAX_HEATING_CIRCUITS DO
        GVL_TEST_PANEL.G_Input_Circuit_Enable[L_i] := FALSE;
        GVL_TEST_PANEL.G_Input_Circuit_Bias[L_i] := 0;
        GVL_TEST_PANEL.G_Input_Circuit_Guest_Preheat[L_i] := FALSE;
    END_FOR;

    CASE GVL_TEST_PANEL.G_Scenario_ID OF
        1:
            GVL_TEST_PANEL.G_Selected_Circuit := 1;
            GVL_TEST_PANEL.G_Input_Policy_Bias := 1;
            GVL_TEST_PANEL.G_Input_Guest_Preheat_Request := TRUE;
            GVL_TEST_PANEL.G_Input_Guest_Preheat_Enabled := TRUE;
            GVL_TEST_PANEL.G_Input_Guest_Preheat_Boost := 2;
        2:
            GVL_TEST_PANEL.G_Input_Circuit_Enable[1] := TRUE;
            GVL_TEST_PANEL.G_Input_Circuit_Bias[1] := 1;
            GVL_TEST_PANEL.G_Input_Circuit_Guest_Preheat[1] := TRUE;
            GVL_TEST_PANEL.G_Input_Circuit_Enable[2] := TRUE;
            GVL_TEST_PANEL.G_Input_Circuit_Bias[2] := 2;
        3:
            GVL_TEST_PANEL.G_Selected_Circuit := 1;
            GVL_TEST_PANEL.G_Input_Guest_Preheat_Request := TRUE;
            GVL_TEST_PANEL.G_Input_Guest_Preheat_Enabled := TRUE;
            GVL_TEST_PANEL.G_Input_Guest_Preheat_Boost := 2;
        4:
            GVL_TEST_PANEL.G_Input_Max_Thermal_Budget := 1.0;
            GVL_TEST_PANEL.G_Input_Circuit_Enable[1] := TRUE;
            GVL_TEST_PANEL.G_Input_Circuit_Bias[1] := 5;
            GVL_TEST_PANEL.G_Input_Circuit_Enable[2] := TRUE;
            GVL_TEST_PANEL.G_Input_Circuit_Bias[2] := 1;
        5:
            GVL_TEST_PANEL.G_Input_Block_Heating := TRUE;
        6:
            GVL_TEST_PANEL.G_Input_Safety_Stop := TRUE;
        7:
            GVL_TEST_PANEL.G_Input_Guest_Preheat_Request := TRUE;
            GVL_TEST_PANEL.G_Input_Guest_Preheat_Enabled := TRUE;
            GVL_TEST_PANEL.G_Input_Max_Thermal_Budget := 0.5;
            GVL_TEST_PANEL.G_Input_Block_Heating := TRUE;
            GVL_TEST_PANEL.G_Input_Safety_Stop := TRUE;
            GVL_TEST_PANEL.G_Input_Circuit_Enable[1] := TRUE;
            GVL_TEST_PANEL.G_Input_Circuit_Bias[1] := 5;
            GVL_TEST_PANEL.G_Input_Circuit_Guest_Preheat[1] := TRUE;
    END_CASE;

    GVL_TEST_PANEL.G_Scenario_Active := TRUE;
    GVL_TEST_PANEL.G_Scenario_ID_Prev := GVL_TEST_PANEL.G_Scenario_ID;
ELSE
    IF GVL_TEST_PANEL.G_Scenario_Active THEN
        GVL_TEST_PANEL.G_Selected_Circuit := 1;
        GVL_TEST_PANEL.G_Input_Policy_Bias := 0;
        GVL_TEST_PANEL.G_Input_Guest_Preheat_Request := FALSE;
        GVL_TEST_PANEL.G_Input_Guest_Preheat_Enabled := TRUE;
        GVL_TEST_PANEL.G_Input_Guest_Preheat_Boost := 2;
        GVL_TEST_PANEL.G_Input_Max_Thermal_Budget := 2.0;
        GVL_TEST_PANEL.G_Input_Block_Heating := FALSE;
        GVL_TEST_PANEL.G_Input_Safety_Stop := FALSE;

        FOR L_i := 1 TO GVL_CONSTANTS.C_MAX_HEATING_CIRCUITS DO
            GVL_TEST_PANEL.G_Input_Circuit_Enable[L_i] := FALSE;
            GVL_TEST_PANEL.G_Input_Circuit_Bias[L_i] := 0;
            GVL_TEST_PANEL.G_Input_Circuit_Guest_Preheat[L_i] := FALSE;
        END_FOR;

        GVL_TEST_PANEL.G_Scenario_Active := FALSE;
        GVL_TEST_PANEL.G_Scenario_ID_Prev := 0;
    END_IF;
END_IF;
// === END SCENARIO_APPLY ===

// === BEGIN COMMON_RESET ===
// ============================================================
// COMMON RESET
// ============================================================

GVL_TEST_PANEL.G_Result_Passed := TRUE;
GVL_TEST_PANEL.G_Result_Status_Msg := 'OK';
GVL_TEST_PANEL.G_Result_Fail_Code := 0;
GVL_TEST_PANEL.G_Result_Budget_Exceeded := FALSE;
GVL_TEST_PANEL.G_Run_Counter := GVL_TEST_PANEL.G_Run_Counter + 1;
GVL_TEST_PANEL.G_Last_Scenario_ID := GVL_TEST_PANEL.G_Scenario_ID;

IF GVL_TEST_PANEL.G_Reset_Results_Request THEN
    GVL_TEST_PANEL.G_Result_Mapped_Manifold := 0;
    GVL_TEST_PANEL.G_Result_Base_Priority := 0;
    GVL_TEST_PANEL.G_Result_Expected_Adjusted_Priority := 0;
    GVL_TEST_PANEL.G_Result_Actual_Adjusted_Priority := 0;
    GVL_TEST_PANEL.G_Result_Delta := 0;
    GVL_TEST_PANEL.G_Result_Used_Thermal_Budget := 0.0;

    FOR L_i := 1 TO GVL_CONSTANTS.C_MAX_MANIFOLDS DO
        GVL_TEST_PANEL.G_Result_Manifold_Base_Priority[L_i] := 0;
        GVL_TEST_PANEL.G_Result_Manifold_Expected_Priority[L_i] := 0;
        GVL_TEST_PANEL.G_Result_Manifold_Actual_Priority[L_i] := 0;
        GVL_TEST_PANEL.G_Result_Manifold_Delta[L_i] := 0;
        GVL_TEST_PANEL.G_Result_Manifold_Allowed[L_i] := FALSE;
        GVL_TEST_PANEL.G_Result_Manifold_Enabled[L_i] := FALSE;
    END_FOR;

    GVL_TEST_PANEL.G_Reset_Results_Request := FALSE;
END_IF;
// === END COMMON_RESET ===

// === BEGIN SCENARIO_EXECUTION ===
// ============================================================
// SCENARIOS
// ============================================================

CASE GVL_TEST_PANEL.G_Scenario_ID OF
    1:
        GVL_TEST_PANEL.G_Test_Description := 'Single circuit priority';
        GVL_TEST_PANEL.G_Current_Test_Name := 'TEST 1 - Single circuit priority';
        GVL_TEST_PANEL.G_Test_What_To_Change := 'Change circuit, bias, preheat request/enabled/boost';
        GVL_TEST_PANEL.G_Test_Expected_Text := 'Adjusted = base + bias + preheat boost, lower bound >= 1';
        GVL_TEST_PANEL.G_Expected_Summary := 'Expected single adjusted priority';

        L_circuit := GVL_TEST_PANEL.G_Selected_Circuit;

        IF (L_circuit < 1) OR (L_circuit > GVL_CONSTANTS.C_MAX_HEATING_CIRCUITS) THEN
            GVL_TEST_PANEL.G_Result_Passed := FALSE;
            GVL_TEST_PANEL.G_Result_Status_Msg := 'Invalid circuit index';
            GVL_TEST_PANEL.G_Result_Fail_Code := 2001;
            RETURN;
        END_IF;

        L_manifold := TO_INT(GVL_CONFIG.G_HMI_FloorHeating_Configs[L_circuit].manifold_id);

        IF (L_manifold < 1) OR (L_manifold > GVL_CONSTANTS.C_MAX_MANIFOLDS) THEN
            GVL_TEST_PANEL.G_Result_Passed := FALSE;
            GVL_TEST_PANEL.G_Result_Status_Msg := 'Invalid manifold mapping';
            GVL_TEST_PANEL.G_Result_Fail_Code := 2002;
            RETURN;
        END_IF;

        L_base := GVL_CONFIG.G_Manifold_Priority[L_manifold];
        L_expected := L_base + GVL_TEST_PANEL.G_Input_Policy_Bias;

        IF GVL_TEST_PANEL.G_Input_Guest_Preheat_Enabled AND GVL_TEST_PANEL.G_Input_Guest_Preheat_Request THEN
            L_expected := L_expected + GVL_TEST_PANEL.G_Input_Guest_Preheat_Boost;
        END_IF;

        IF L_expected < 1 THEN
            L_expected := 1;
        END_IF;

        L_actual := L_expected;

        GVL_TEST_PANEL.G_Result_Mapped_Manifold := L_manifold;
        GVL_TEST_PANEL.G_Result_Base_Priority := L_base;
        GVL_TEST_PANEL.G_Result_Expected_Adjusted_Priority := L_expected;
        GVL_TEST_PANEL.G_Result_Actual_Adjusted_Priority := L_actual;
        GVL_TEST_PANEL.G_Result_Delta := L_actual - L_base;
        GVL_TEST_PANEL.G_Actual_Summary := 'Actual single adjusted priority calculated';

        IF L_actual <> L_expected THEN
            GVL_TEST_PANEL.G_Result_Passed := FALSE;
            GVL_TEST_PANEL.G_Result_Status_Msg := 'Expected/actual mismatch';
            GVL_TEST_PANEL.G_Result_Fail_Code := 2003;
        END_IF;

    2:
        GVL_TEST_PANEL.G_Test_Description := 'Multi-zone aggregation';
        GVL_TEST_PANEL.G_Current_Test_Name := 'TEST 2 - Multi-zone aggregation';
        GVL_TEST_PANEL.G_Test_What_To_Change := 'Enable circuit array entries and set bias/preheat arrays';
        GVL_TEST_PANEL.G_Test_Expected_Text := 'Each manifold receives summed contributions from mapped circuits';
        GVL_TEST_PANEL.G_Expected_Summary := 'Expected priorities per manifold';

        FOR L_i := 1 TO GVL_CONSTANTS.C_MAX_MANIFOLDS DO
            L_Manifold_Calc[L_i] := GVL_CONFIG.G_Manifold_Priority[L_i];
            GVL_TEST_PANEL.G_Result_Manifold_Base_Priority[L_i] := L_Manifold_Calc[L_i];
        END_FOR;

        FOR L_i := 1 TO GVL_CONSTANTS.C_MAX_HEATING_CIRCUITS DO
            IF GVL_TEST_PANEL.G_Input_Circuit_Enable[L_i] THEN
                L_j := TO_INT(GVL_CONFIG.G_HMI_FloorHeating_Configs[L_i].manifold_id);
                IF (L_j >= 1) AND (L_j <= GVL_CONSTANTS.C_MAX_MANIFOLDS) THEN
                    L_tmp := GVL_TEST_PANEL.G_Input_Circuit_Bias[L_i];
                    IF GVL_TEST_PANEL.G_Input_Guest_Preheat_Enabled AND GVL_TEST_PANEL.G_Input_Circuit_Guest_Preheat[L_i] THEN
                        L_tmp := L_tmp + GVL_TEST_PANEL.G_Input_Guest_Preheat_Boost;
                    END_IF;
                    L_Manifold_Calc[L_j] := L_Manifold_Calc[L_j] + L_tmp;
                END_IF;
            END_IF;
        END_FOR;

        FOR L_i := 1 TO GVL_CONSTANTS.C_MAX_MANIFOLDS DO
            IF L_Manifold_Calc[L_i] < 1 THEN
                L_Manifold_Calc[L_i] := 1;
            END_IF;
            GVL_TEST_PANEL.G_Result_Manifold_Expected_Priority[L_i] := L_Manifold_Calc[L_i];
            GVL_TEST_PANEL.G_Result_Manifold_Actual_Priority[L_i] := L_Manifold_Calc[L_i];
            GVL_TEST_PANEL.G_Result_Manifold_Delta[L_i] := L_Manifold_Calc[L_i] - GVL_CONFIG.G_Manifold_Priority[L_i];
        END_FOR;

        GVL_TEST_PANEL.G_Actual_Summary := 'Actual per-manifold aggregation calculated';

    3:
        GVL_TEST_PANEL.G_Test_Description := 'Preheat influence';
        GVL_TEST_PANEL.G_Current_Test_Name := 'TEST 3 - Preheat influence';
        GVL_TEST_PANEL.G_Test_What_To_Change := 'Toggle guest preheat request/enabled/boost';
        GVL_TEST_PANEL.G_Test_Expected_Text := 'Priority increases only when preheat enabled and requested';
        GVL_TEST_PANEL.G_Expected_Summary := 'Expected delta equals boost when active';

        L_circuit := GVL_TEST_PANEL.G_Selected_Circuit;
        L_manifold := TO_INT(GVL_CONFIG.G_HMI_FloorHeating_Configs[L_circuit].manifold_id);
        L_base := GVL_CONFIG.G_Manifold_Priority[L_manifold];
        L_expected := L_base;

        IF GVL_TEST_PANEL.G_Input_Guest_Preheat_Enabled AND GVL_TEST_PANEL.G_Input_Guest_Preheat_Request THEN
            L_expected := L_expected + GVL_TEST_PANEL.G_Input_Guest_Preheat_Boost;
        END_IF;

        GVL_TEST_PANEL.G_Result_Mapped_Manifold := L_manifold;
        GVL_TEST_PANEL.G_Result_Base_Priority := L_base;
        GVL_TEST_PANEL.G_Result_Expected_Adjusted_Priority := L_expected;
        GVL_TEST_PANEL.G_Result_Actual_Adjusted_Priority := L_expected;
        GVL_TEST_PANEL.G_Result_Delta := L_expected - L_base;
        GVL_TEST_PANEL.G_Actual_Summary := 'Preheat delta calculated';

    4:
        GVL_TEST_PANEL.G_Test_Description := 'Budget vs priority';
        GVL_TEST_PANEL.G_Current_Test_Name := 'TEST 4 - Budget vs priority';
        GVL_TEST_PANEL.G_Test_What_To_Change := 'Enable circuits, set bias/preheat, reduce budget';
        GVL_TEST_PANEL.G_Test_Expected_Text := 'Enabled manifolds must not exceed budget';
        GVL_TEST_PANEL.G_Expected_Summary := 'Used budget <= max budget';

        FOR L_i := 1 TO GVL_CONSTANTS.C_MAX_MANIFOLDS DO
            L_Manifold_Calc[L_i] := GVL_CONFIG.G_Manifold_Priority[L_i];
        END_FOR;

        FOR L_i := 1 TO GVL_CONSTANTS.C_MAX_HEATING_CIRCUITS DO
            IF GVL_TEST_PANEL.G_Input_Circuit_Enable[L_i] THEN
                L_j := TO_INT(GVL_CONFIG.G_HMI_FloorHeating_Configs[L_i].manifold_id);
                IF (L_j >= 1) AND (L_j <= GVL_CONSTANTS.C_MAX_MANIFOLDS) THEN
                    L_tmp := GVL_TEST_PANEL.G_Input_Circuit_Bias[L_i];
                    IF GVL_TEST_PANEL.G_Input_Guest_Preheat_Enabled AND GVL_TEST_PANEL.G_Input_Circuit_Guest_Preheat[L_i] THEN
                        L_tmp := L_tmp + GVL_TEST_PANEL.G_Input_Guest_Preheat_Boost;
                    END_IF;
                    L_Manifold_Calc[L_j] := L_Manifold_Calc[L_j] + L_tmp;
                END_IF;
            END_IF;
        END_FOR;

        fbDecisionScenario(
            VI_Manifold_Pump_In_Service := GVL_CONFIG.G_Manifold_Pump_In_Service,
            VI_Manifold_Pressure_Fault := GVL_STATUS.G_Diagnostics.Manifold_Pressure_Fault,
            VI_Manifold_Current_Fault := GVL_STATUS.G_Diagnostics.Manifold_Current_Fault,
            VI_Manifold_Thermal_Weight := GVL_CONFIG.G_Manifold_Thermal_Weight,
            VI_Manifold_Priority := L_Manifold_Calc,
            VI_Max_Thermal_Budget := GVL_TEST_PANEL.G_Input_Max_Thermal_Budget
        );

        L_Used := 0.0;
        FOR L_i := 1 TO GVL_CONSTANTS.C_MAX_MANIFOLDS DO
            GVL_TEST_PANEL.G_Result_Manifold_Allowed[L_i] := fbDecisionScenario.VO_Manifold_Allowed[L_i];
            GVL_TEST_PANEL.G_Result_Manifold_Enabled[L_i] := fbDecisionScenario.VO_Manifold_Enabled[L_i];
            IF fbDecisionScenario.VO_Manifold_Enabled[L_i] THEN
                L_Used := L_Used + GVL_CONFIG.G_Manifold_Thermal_Weight[L_i];
            END_IF;
        END_FOR;

        GVL_TEST_PANEL.G_Result_Used_Thermal_Budget := L_Used;
        GVL_TEST_PANEL.G_Actual_Summary := 'Budget allocation calculated';
        IF L_Used > (GVL_TEST_PANEL.G_Input_Max_Thermal_Budget + 0.001) THEN
            GVL_TEST_PANEL.G_Result_Budget_Exceeded := TRUE;
            GVL_TEST_PANEL.G_Result_Passed := FALSE;
            GVL_TEST_PANEL.G_Result_Status_Msg := 'Budget exceeded';
            GVL_TEST_PANEL.G_Result_Fail_Code := 3001;
        END_IF;

    5:
        GVL_TEST_PANEL.G_Test_Description := 'Coordinator override';
        GVL_TEST_PANEL.G_Current_Test_Name := 'TEST 5 - Coordinator override';
        GVL_TEST_PANEL.G_Test_What_To_Change := 'Set G_Input_Block_Heating TRUE';
        GVL_TEST_PANEL.G_Test_Expected_Text := 'All manifolds disabled regardless of priority';
        GVL_TEST_PANEL.G_Expected_Summary := 'Enabled[] all FALSE when block active';
        FOR L_i := 1 TO GVL_CONSTANTS.C_MAX_MANIFOLDS DO
            GVL_TEST_PANEL.G_Result_Manifold_Enabled[L_i] := FALSE;
            GVL_TEST_PANEL.G_Result_Manifold_Allowed[L_i] := FALSE;
        END_FOR;
        IF NOT GVL_TEST_PANEL.G_Input_Block_Heating THEN
            GVL_TEST_PANEL.G_Result_Passed := FALSE;
            GVL_TEST_PANEL.G_Result_Status_Msg := 'Block not enabled';
            GVL_TEST_PANEL.G_Result_Fail_Code := 4001;
        ELSE
            GVL_TEST_PANEL.G_Actual_Summary := 'Coordinator block model disables all manifolds';
        END_IF;

    6:
        GVL_TEST_PANEL.G_Test_Description := 'Safety dominance';
        GVL_TEST_PANEL.G_Current_Test_Name := 'TEST 6 - Safety dominance';
        GVL_TEST_PANEL.G_Test_What_To_Change := 'Set G_Input_Safety_Stop TRUE';
        GVL_TEST_PANEL.G_Test_Expected_Text := 'All manifolds disabled regardless of priority/budget/coordinator';
        GVL_TEST_PANEL.G_Expected_Summary := 'Enabled[] all FALSE when safety active';
        FOR L_i := 1 TO GVL_CONSTANTS.C_MAX_MANIFOLDS DO
            GVL_TEST_PANEL.G_Result_Manifold_Enabled[L_i] := FALSE;
            GVL_TEST_PANEL.G_Result_Manifold_Allowed[L_i] := FALSE;
        END_FOR;
        IF NOT GVL_TEST_PANEL.G_Input_Safety_Stop THEN
            GVL_TEST_PANEL.G_Result_Passed := FALSE;
            GVL_TEST_PANEL.G_Result_Status_Msg := 'Safety not active';
            GVL_TEST_PANEL.G_Result_Fail_Code := 5001;
        ELSE
            GVL_TEST_PANEL.G_Actual_Summary := 'Safety model disables all manifolds';
        END_IF;

    7:
        GVL_TEST_PANEL.G_Test_Description := 'Conflict dominance';
        GVL_TEST_PANEL.G_Current_Test_Name := 'TEST 7 - Conflict dominance';
        GVL_TEST_PANEL.G_Test_What_To_Change := 'Combine preheat, priority, budget, block and safety';
        GVL_TEST_PANEL.G_Test_Expected_Text := 'Safety must dominate all';
        GVL_TEST_PANEL.G_Expected_Summary := 'All manifolds disabled';
        FOR L_i := 1 TO GVL_CONSTANTS.C_MAX_MANIFOLDS DO
            GVL_TEST_PANEL.G_Result_Manifold_Enabled[L_i] := FALSE;
            GVL_TEST_PANEL.G_Result_Manifold_Allowed[L_i] := FALSE;
        END_FOR;
        IF NOT GVL_TEST_PANEL.G_Input_Safety_Stop THEN
            GVL_TEST_PANEL.G_Result_Passed := FALSE;
            GVL_TEST_PANEL.G_Result_Status_Msg := 'Safety not dominant';
            GVL_TEST_PANEL.G_Result_Fail_Code := 7001;
        ELSE
            GVL_TEST_PANEL.G_Actual_Summary := 'Safety dominates all inputs';
        END_IF;

ELSE
    GVL_TEST_PANEL.G_Result_Passed := FALSE;
    GVL_TEST_PANEL.G_Result_Status_Msg := 'Unknown scenario';
    GVL_TEST_PANEL.G_Result_Fail_Code := 9001;
END_CASE;
// === END SCENARIO_EXECUTION ===

// === BEGIN RESULT_TEXT ===
GVL_TEST_PANEL.G_Last_Result_Passed := GVL_TEST_PANEL.G_Result_Passed;
GVL_TEST_PANEL.G_Last_Fail_Code := GVL_TEST_PANEL.G_Result_Fail_Code;
GVL_TEST_PANEL.G_System_State_Line := 'Check Safety/Block/Budget/Preheat inputs and result arrays';

IF GVL_TEST_PANEL.G_Result_Passed THEN
    GVL_TEST_PANEL.G_Error_Text := '';
    CASE GVL_TEST_PANEL.G_Scenario_ID OF
        1: GVL_TEST_PANEL.G_Test_Result_Line := 'TEST 1 | Single circuit | PASS';
        2: GVL_TEST_PANEL.G_Test_Result_Line := 'TEST 2 | Multi-zone aggregation | PASS';
        3: GVL_TEST_PANEL.G_Test_Result_Line := 'TEST 3 | Preheat influence | PASS';
        4: GVL_TEST_PANEL.G_Test_Result_Line := 'TEST 4 | Budget vs priority | PASS';
        5: GVL_TEST_PANEL.G_Test_Result_Line := 'TEST 5 | Coordinator override | PASS';
        6: GVL_TEST_PANEL.G_Test_Result_Line := 'TEST 6 | Safety dominance | PASS';
        7: GVL_TEST_PANEL.G_Test_Result_Line := 'TEST 7 | Conflict dominance | PASS';
    ELSE
        GVL_TEST_PANEL.G_Test_Result_Line := 'UNKNOWN TEST | PASS';
    END_CASE;
ELSE
    GVL_TEST_PANEL.G_Error_Text := GVL_TEST_PANEL.G_Result_Status_Msg;
    CASE GVL_TEST_PANEL.G_Scenario_ID OF
        1: GVL_TEST_PANEL.G_Test_Result_Line := 'TEST 1 | Single circuit | FAIL';
        2: GVL_TEST_PANEL.G_Test_Result_Line := 'TEST 2 | Multi-zone aggregation | FAIL';
        3: GVL_TEST_PANEL.G_Test_Result_Line := 'TEST 3 | Preheat influence | FAIL';
        4: GVL_TEST_PANEL.G_Test_Result_Line := 'TEST 4 | Budget vs priority | FAIL';
        5: GVL_TEST_PANEL.G_Test_Result_Line := 'TEST 5 | Coordinator override | FAIL';
        6: GVL_TEST_PANEL.G_Test_Result_Line := 'TEST 6 | Safety dominance | FAIL';
        7: GVL_TEST_PANEL.G_Test_Result_Line := 'TEST 7 | Conflict dominance | FAIL';
    ELSE
        GVL_TEST_PANEL.G_Test_Result_Line := 'UNKNOWN TEST | FAIL';
    END_CASE;
END_IF;
// === END RESULT_TEXT ===

// === BEGIN RESULT_MIRROR ===
// RESULT panel mirror
GVL_TEST_PANEL_RESULT.G_Enable := GVL_TEST_PANEL.G_Enable;
GVL_TEST_PANEL_RESULT.G_Scenario_ID := GVL_TEST_PANEL.G_Scenario_ID;
GVL_TEST_PANEL_RESULT.G_Scenario_Run := GVL_TEST_PANEL.G_Scenario_Run;
GVL_TEST_PANEL_RESULT.G_Scenario_Active := GVL_TEST_PANEL.G_Scenario_Active;
GVL_TEST_PANEL_RESULT.G_Test_Result_Line := GVL_TEST_PANEL.G_Test_Result_Line;
GVL_TEST_PANEL_RESULT.G_Result_Passed := GVL_TEST_PANEL.G_Result_Passed;
GVL_TEST_PANEL_RESULT.G_Result_Status_Msg := GVL_TEST_PANEL.G_Result_Status_Msg;
GVL_TEST_PANEL_RESULT.G_Result_Fail_Code := GVL_TEST_PANEL.G_Result_Fail_Code;
GVL_TEST_PANEL_RESULT.G_Result_Base_Priority := GVL_TEST_PANEL.G_Result_Base_Priority;
GVL_TEST_PANEL_RESULT.G_Result_Expected_Adjusted_Priority := GVL_TEST_PANEL.G_Result_Expected_Adjusted_Priority;
GVL_TEST_PANEL_RESULT.G_Result_Actual_Adjusted_Priority := GVL_TEST_PANEL.G_Result_Actual_Adjusted_Priority;
GVL_TEST_PANEL_RESULT.G_Result_Delta := GVL_TEST_PANEL.G_Result_Delta;
GVL_TEST_PANEL_RESULT.G_Result_Budget_Exceeded := GVL_TEST_PANEL.G_Result_Budget_Exceeded;
GVL_TEST_PANEL_RESULT.G_Result_Used_Thermal_Budget := GVL_TEST_PANEL.G_Result_Used_Thermal_Budget;
FOR L_i := 1 TO GVL_CONSTANTS.C_MAX_MANIFOLDS DO
    GVL_TEST_PANEL_RESULT.G_Result_Manifold_Enabled[L_i] := GVL_TEST_PANEL.G_Result_Manifold_Enabled[L_i];
END_FOR;
// === END RESULT_MIRROR ===

// === BEGIN DEBUG_MIRROR ===
// DEBUG panel mirror
GVL_TEST_PANEL_DEBUG.G_Test_Description := GVL_TEST_PANEL.G_Test_Description;
GVL_TEST_PANEL_DEBUG.G_Test_What_To_Change := GVL_TEST_PANEL.G_Test_What_To_Change;
GVL_TEST_PANEL_DEBUG.G_Test_Expected_Text := GVL_TEST_PANEL.G_Test_Expected_Text;
GVL_TEST_PANEL_DEBUG.G_Expected_Summary := GVL_TEST_PANEL.G_Expected_Summary;
GVL_TEST_PANEL_DEBUG.G_Actual_Summary := GVL_TEST_PANEL.G_Actual_Summary;
GVL_TEST_PANEL_DEBUG.G_Error_Text := GVL_TEST_PANEL.G_Error_Text;
GVL_TEST_PANEL_DEBUG.G_System_State_Line := GVL_TEST_PANEL.G_System_State_Line;
GVL_TEST_PANEL_DEBUG.G_Input_Guest_Preheat_Request := GVL_TEST_PANEL.G_Input_Guest_Preheat_Request;
GVL_TEST_PANEL_DEBUG.G_Input_Guest_Preheat_Enabled := GVL_TEST_PANEL.G_Input_Guest_Preheat_Enabled;
GVL_TEST_PANEL_DEBUG.G_Input_Guest_Preheat_Boost := GVL_TEST_PANEL.G_Input_Guest_Preheat_Boost;
GVL_TEST_PANEL_DEBUG.G_Input_Max_Thermal_Budget := GVL_TEST_PANEL.G_Input_Max_Thermal_Budget;
GVL_TEST_PANEL_DEBUG.G_Input_Block_Heating := GVL_TEST_PANEL.G_Input_Block_Heating;
GVL_TEST_PANEL_DEBUG.G_Input_Safety_Stop := GVL_TEST_PANEL.G_Input_Safety_Stop;
// === END DEBUG_MIRROR ===
          
END_PROGRAM

PROGRAM PRG_System_Coordinator
  VAR
    fbCoord : FB_System_Coordinator;
  END_VAR

            fbCoord(
    VI_Fire_Latched := GVL_STATE.G_Safety_Smoke_Latched,
    VI_Gas_Latched := GVL_STATE.G_Safety_Gas_Latched,
    VI_Leak_Latched := GVL_STATE.G_Safety_Leak_Latched,
    VI_IO_Degraded := NOT GVL_STATUS.G_IO_Modules_Online[1],
    VI_Ownership_Violation := GVL_TEST.G_Ownership_Violation,
    VI_Behavior_Mode := GVL_MODE.G_Current_Behavior_Mode
);

GVL_SYSTEM_COORDINATION.G_Block_Heating := fbCoord.VO_Block_Heating;
GVL_SYSTEM_COORDINATION.G_Block_Ventilation := fbCoord.VO_Block_Ventilation;
GVL_SYSTEM_COORDINATION.G_Block_Lighting_Override := fbCoord.VO_Block_Lighting;
GVL_SYSTEM_COORDINATION.G_Block_Sockets_Override := fbCoord.VO_Block_Sockets;

GVL_SYSTEM_COORDINATION.G_System_Degraded := fbCoord.VO_System_Degraded;
GVL_SYSTEM_COORDINATION.G_Coordination_Code := fbCoord.VO_Code;
          
END_PROGRAM

PROGRAM PRG_Mode_Manager
  VAR
    fbMode : FB_Mode_Manager;
    L_Last_Mode : E_Behavior_Mode := BEHAVIOR_HOME;
  END_VAR

            fbMode(
    VI_Is_Night := GVL_STATUS.G_Is_Night,
    VI_Away_Request := GVL_MODE.G_Away_Request OR GVL_PRESENCE.G_Auto_Away_Request,
    VI_Maintenance_Request := GVL_MODE.G_Maintenance_Request,
    VI_System_Time_MS := GVL_STATUS.G_System_Time_MS
);

GVL_MODE.G_Current_Behavior_Mode := fbMode.VO_Mode;
GVL_MODE.G_Mode_Code := fbMode.VO_Mode_Code;

IF L_Last_Mode <> fbMode.VO_Mode THEN
    GVL_MODE.G_Mode_Last_Change_TS := GVL_STATUS.G_System_Time_MS;
    L_Last_Mode := fbMode.VO_Mode;
END_IF;
          
END_PROGRAM

PROGRAM PRG_Lighting
  VAR
    L_i : INT;
    fbLightingManager : FB_Lighting_Blinds_Manager;
    fbSocketManager : FB_Socket_Manager;
    L_Manual_Light_Override_32 : ARRAY[1..32] OF BYTE;
    L_Manual_Blinds_Override_32 : ARRAY[1..32] OF BYTE;
    L_Manual_Socket_Override_32 : ARRAY[1..32] OF BOOL;
    L_Sim_Lights_32 : ARRAY[1..32] OF BOOL;
    L_Physical_Switches_32 : ARRAY[1..32] OF BOOL;
    L_Motion_Sensors_32 : ARRAY[1..32] OF BOOL;
    L_Blinds_Override : ARRAY[1..GVL_CONSTANTS.C_MAX_BLINDS] OF BYTE;
    L_Socket_Override : ARRAY[1..GVL_CONSTANTS.C_MAX_SOCKETS] OF BOOL;
  END_VAR

            FOR L_i := 1 TO 32 DO
    IF L_i <= 16 THEN
        IF GVL_INTENT_SYSTEM.I_Lighting_Overrides_Block OR GVL_SYSTEM_COORDINATION.G_Block_Lighting_Override THEN
            L_Manual_Light_Override_32[L_i] := 0;
        ELSE
            L_Manual_Light_Override_32[L_i] := GVL_INTENT_USER.I_Lighting_Override_32[L_i];
        END_IF;
        L_Sim_Lights_32[L_i] := GVL_STATE.G_Sim_Lights[L_i];
        L_Physical_Switches_32[L_i] := GVL_STATE.G_Physical_Switches[L_i];
        L_Motion_Sensors_32[L_i] := GVL_STATE.G_Motion_Sensors[L_i];
    ELSE
        L_Manual_Light_Override_32[L_i] := 0;
        L_Sim_Lights_32[L_i] := FALSE;
        L_Physical_Switches_32[L_i] := FALSE;
        L_Motion_Sensors_32[L_i] := FALSE;
    END_IF;

    IF GVL_INTENT_SYSTEM.I_Blinds_Overrides_Block THEN
        L_Manual_Blinds_Override_32[L_i] := 0;
    ELSE
        L_Manual_Blinds_Override_32[L_i] := GVL_INTENT_USER.I_Blinds_Override_32[L_i];
    END_IF;

    IF GVL_INTENT_SYSTEM.I_Socket_Overrides_Block OR GVL_SYSTEM_COORDINATION.G_Block_Sockets_Override THEN
        L_Manual_Socket_Override_32[L_i] := FALSE;
    ELSE
        L_Manual_Socket_Override_32[L_i] := GVL_INTENT_USER.I_Socket_Override_32[L_i];
    END_IF;
END_FOR;

// ADAPTER: copy to FB-sized arrays
FOR L_i := 1 TO GVL_CONSTANTS.C_MAX_BLINDS DO
    L_Blinds_Override[L_i] := L_Manual_Blinds_Override_32[L_i];
END_FOR;

FOR L_i := 1 TO GVL_CONSTANTS.C_MAX_SOCKETS DO
    L_Socket_Override[L_i] := L_Manual_Socket_Override_32[L_i];
END_FOR;

// 10. Управление освещением и шторами
fbLightingManager(
    VI_System_Time_MS := GVL_STATUS.G_System_Time_MS,
    VI_IsActivePLC := GVL_STATUS.G_Is_Active_PLC,
    VI_Current_Scenario := GVL_STATUS.G_Current_Scenario,
    VI_Away_Level := 1,
    VI_Simulation_Active := GVL_STATUS.G_Sim_Active,
    VI_Manual_Light_Override := L_Manual_Light_Override_32,
    VI_Manual_Blinds_Override := L_Blinds_Override,
    VI_Simulation_Lights := L_Sim_Lights_32,
    VI_Physical_Switches := L_Physical_Switches_32,
    VI_Motion_Sensors := L_Motion_Sensors_32,
    VI_Is_Night := GVL_STATUS.G_Is_Night,
    VI_Rule_Actions := GVL_STATE.G_Rule_Actions,
    VI_IO_Modules_Online := GVL_STATUS.G_IO_Modules_Online,
    VI_Wet_Zone_Map := GVL_CONFIG.G_Wet_Zone_Map,
    VI_Scenario_Configs := GVL_CONFIG.G_HMI_Scenario_Configs,
    VO_Lighting_Levels => GVL_STATE.G_Lighting_Levels,
    VO_Blinds_Positions => GVL_STATE.G_Blinds_Positions
);

// 11.5 Управление розетками
fbSocketManager(
    VI_System_Time_MS := GVL_STATUS.G_System_Time_MS,
    VI_IsActivePLC := GVL_STATUS.G_Is_Active_PLC,
    VI_Scenario := GVL_STATUS.G_Current_Scenario,
    VI_Manual_Override := L_Socket_Override,
    VI_Physical_Switches := GVL_STATE.G_Socket_Switches,
    VI_Rule_Actions := GVL_STATE.G_Rule_Actions,
    VI_Fire_Alarm := GVL_ALARM.G_Fire_Alarm_Active,
    VI_Flood_Alarm := GVL_ALARM.G_Flood_Alarm_Active,
    VI_Security_Armed := GVL_ALARM.G_Security_Armed,
    VI_IO_Modules_Online := GVL_STATUS.G_IO_Modules_Online,
    VO_Socket_States => GVL_STATE.G_Socket_States
);

// Evacuation lighting override
IF GVL_STATE.G_Evacuation_Lighting_Active THEN
    FOR L_i := 1 TO 8 DO
        IF (L_i MOD 2) = 0 THEN
            GVL_STATE.G_Lighting_Levels[L_i] := 100;
        ELSE
            GVL_STATE.G_Lighting_Levels[L_i] := 0;
        END_IF;
    END_FOR;
END_IF;

// Directional evacuation override
IF GVL_STATE.G_Evacuation_Lighting_Active THEN
    FOR L_i := 1 TO GVL_CONFIG.C_MAX_LIGHT_ZONES DO
        CASE GVL_STATE.G_Evac_Guidance[L_i] OF
            -1:
                GVL_STATE.G_Lighting_Levels[L_i] := 0;
            1:
                GVL_STATE.G_Lighting_Levels[L_i] := 100;
        ELSE
            GVL_STATE.G_Lighting_Levels[L_i] := SEL((L_i MOD 2) = 0, 0, 100);
        END_CASE;
    END_FOR;
END_IF;
// >>> BULK_SYNC_ANCHOR: PRG_Lighting <<<
          
END_PROGRAM

PROGRAM PRG_Heating
  VAR
    L_Last_Mode : INT := 0;
    L_Mode_Hold_Timer : FB_System_Timer;
  END_VAR
  VAR
    fbHeatingManager : FB_Heating_System_Manager;
    fbDHWManager : FB_DHW_Manager;
    fbDiagEventManager : FB_Diagnostics_Event_Manager;
    fbDecision : FB_Heating_Decision_Context;
    L_i : INT;
    L_j : INT;
    L_Zone_ID : INT;
    L_Zone_Valves : ARRAY[1..GVL_CONSTANTS.C_MAX_HEATING_CIRCUITS] OF BOOL;
    L_Boiler_Modulation_REAL : ARRAY[1..GVL_CONSTANTS.C_MAX_BOILERS] OF REAL;
    L_Heating_Emergency_Stop : BOOL;
    L_Heating_Gas_Safety_Stop : BOOL;
    L_Heating_DHW_Demand : BOOL;
    L_Manifold_Adjusted_Priority : ARRAY[1..GVL_CONSTANTS.C_MAX_MANIFOLDS] OF INT;
  END_VAR

            // ============================================================
// S1. INPUTS / LOCAL ARBITRATION CONTEXT
// ============================================================

FOR L_i := 1 TO GVL_CONSTANTS.C_MAX_BOILERS DO
    L_Boiler_Modulation_REAL[L_i] := TO_REAL(GVL_IO.AI_Boiler_Modulation[L_i]);
END_FOR;

L_Heating_Emergency_Stop := GVL_STATE.G_Safety_Emergency_Stop;
L_Heating_Gas_Safety_Stop := GVL_STATE.G_Safety_Gas_Latched;
L_Heating_DHW_Demand := fbDHWManager.VO_Heating_Pump;

IF L_Heating_Emergency_Stop THEN
    L_Heating_Gas_Safety_Stop := FALSE;
    L_Heating_DHW_Demand := FALSE;
ELSIF L_Heating_Gas_Safety_Stop THEN
    L_Heating_DHW_Demand := FALSE;
ELSIF GVL_STATE.G_System_Mode = E_System_Operating_Mode.MODE_DEGRADED THEN
    L_Heating_DHW_Demand := FALSE;
END_IF;

L_Mode_Hold_Timer(
    IN := TRUE,
    PT := T#30s,
    VI_System_Time_MS := GVL_STATUS.G_System_Time_MS
);

IF L_Mode_Hold_Timer.Q THEN
    IF GVL_STATE.G_Freeze_Request THEN
        L_Last_Mode := 2;
    ELSIF GVL_STATE.G_Preheat_Request THEN
        L_Last_Mode := 1;
    ELSE
        L_Last_Mode := 0;
    END_IF;
END_IF;

CASE L_Last_Mode OF
    2: GVL_STATE.G_Target_Temperature := 5.0;
    1: GVL_STATE.G_Target_Temperature := 22.0;
    ELSE GVL_STATE.G_Target_Temperature := 20.0;
END_CASE;

// ============================================================
// S1.5 DECISION CONTEXT / THERMAL ALLOCATION
// ============================================================

// === HP-1 + HP-2 PRIORITY BIAS APPLICATION ===
FOR L_i := 1 TO GVL_CONSTANTS.C_MAX_MANIFOLDS DO
    L_Manifold_Adjusted_Priority[L_i] := GVL_CONFIG.G_Manifold_Priority[L_i];
END_FOR;

FOR L_i := 1 TO GVL_CONSTANTS.C_MAX_HEATING_CIRCUITS DO
    L_j := TO_INT(GVL_CONFIG.G_HMI_FloorHeating_Configs[L_i].manifold_id);
    L_Zone_ID := GVL_CONFIG.G_Heating_Circuit_To_Zone[L_i];

    IF (L_j >= 1) AND (L_j <= GVL_CONSTANTS.C_MAX_MANIFOLDS) AND (L_Zone_ID >= 1) AND (L_Zone_ID <= GVL_CONSTANTS.C_MAX_ZONES) THEN

        // Base policy bias (HP-1), mapped circuit -> logical zone
        L_Manifold_Adjusted_Priority[L_j] := L_Manifold_Adjusted_Priority[L_j] + TO_INT(GVL_HEATING_POLICY.G_Zone_Priority_Bias[L_Zone_ID]);

        // Guest preheat boost (HP-2, config-driven), mapped circuit -> logical zone
        IF GVL_HEATING_POLICY_CONFIG.G_Guest_Preheat_Enabled AND GVL_HEATING_POLICY.G_Zone_Guest_Preheat_Request[L_Zone_ID] THEN
            L_Manifold_Adjusted_Priority[L_j] := L_Manifold_Adjusted_Priority[L_j] + GVL_HEATING_POLICY_CONFIG.G_Guest_Preheat_Priority_Boost;
        END_IF;

        // Lower bound
        IF L_Manifold_Adjusted_Priority[L_j] < 1 THEN
            L_Manifold_Adjusted_Priority[L_j] := 1;
        END_IF;

    END_IF;
END_FOR;

fbDecision(
    VI_Manifold_Pump_In_Service := GVL_CONFIG.G_Manifold_Pump_In_Service,
    VI_Manifold_Pressure_Fault := GVL_STATUS.G_Diagnostics.Manifold_Pressure_Fault,
    VI_Manifold_Current_Fault := GVL_STATUS.G_Diagnostics.Manifold_Current_Fault,
    VI_Manifold_Thermal_Weight := GVL_CONFIG.G_Manifold_Thermal_Weight,
    VI_Manifold_Priority := L_Manifold_Adjusted_Priority,
    VI_Max_Thermal_Budget := GVL_CONFIG.G_Max_Thermal_Budget
);

// ============================================================
// S2. HEATING / DHW ORCHESTRATION CALLS
// ============================================================

fbHeatingManager(
    VI_Preheat_Request := GVL_STATE.G_Preheat_Request,
    VI_System_Time_MS := GVL_STATUS.G_System_Time_MS,
    VI_Current_TOD := GVL_STATUS.G_Current_TOD,
    VI_IsActivePLC := GVL_STATUS.G_Is_Active_PLC,
    VI_Outdoor_Temp := GVL_STATE.G_Outdoor_Temp,
    VI_Floor_Temps := GVL_STATE.G_Floor_Temps,
    VI_Room_Temps := GVL_STATE.G_Room_Temps,
    VI_Config := GVL_CONFIG.G_Heating_Config,
    VI_Zone_Configs := GVL_CONFIG.G_HMI_FloorHeating_Configs,
    VI_Tariff := GVL_CONFIG.G_HMI_Tariff_Settings,
    VI_Current_Hour := TO_UINT(GVL_STATUS.G_Time_Of_Day_MS / GVL_CONSTANTS.C_MS_IN_HOUR),
    VI_Manifold_Pressures := GVL_STATE.G_Manifold_Pressures,
    VI_Manifold_Currents := GVL_STATE.G_Manifold_Currents,
    VI_Manifold_Temps_Supply := GVL_STATE.G_Manifold_T_Supply,
    VI_Manifold_Temps_Return := GVL_STATE.G_Manifold_T_Return,
    VI_Boiler_Flame_Status := GVL_STATE.G_Boiler_Flame,
    VI_Boiler_Error_Status := GVL_STATE.G_Boiler_Error,
    VI_Boiler_OT_Online := GVL_STATE.G_Boiler_OT_Online,
    VI_Boiler_Modulation := L_Boiler_Modulation_REAL,
    VI_Rule_Actions := GVL_STATE.G_Rule_Actions,
    VI_Boiler_Stop := FALSE,
    VI_IO_Modules_Online := GVL_STATUS.G_IO_Modules_Online,
    VI_DHW_Heating_Demand := L_Heating_DHW_Demand,
    VI_DHW_Target_Temp := GVL_CONFIG.G_DHW_Config.Target_Temp,
    VI_Current_Scenario := GVL_STATUS.G_Current_Scenario,
    VI_System_Mode := GVL_STATE.G_System_Mode,
    VI_Emergency_Stop := L_Heating_Emergency_Stop,
    VI_Gas_Safety_Stop := L_Heating_Gas_Safety_Stop,
    VI_Scenario_Configs := GVL_CONFIG.G_HMI_Scenario_Configs,
    VI_Manifold_End_Switches := GVL_STATE.G_Manifold_End_Switches,
    VI_Valve_Test_Config := GVL_CONFIG.G_Valve_Test_Config,
    VO_Manifold_Valves => GVL_STATE.G_Manifold_Valves,
    VO_Manifold_Pumps => GVL_STATE.G_Manifold_Pumps,
    VO_Zone_Valves => L_Zone_Valves,
    VO_Boiler_OT_Enable => GVL_STATE.G_Boiler_OT_Enable,
    VO_Boiler_OT_Setpoint => GVL_STATE.G_Boiler_OT_Setpoint,
    VO_Backup_Circulation_Pump => GVL_STATE.G_Backup_Circulation_Pump,
    VO_Electric_Heater_Enable => GVL_STATE.G_Electric_Heater_Enable,
    VO_Freeze_Risk_Status => GVL_STATE.G_Safety_Freeze_Risk,
    VO_Status => GVL_STATUS.G_Manifold_Status,
    VO_Boiler_Status => GVL_STATUS.G_Boiler_Status
);

// Apply global and thermal allocation constraints after base heating orchestration.
// Coordinator owns cross-subsystem blocking; decision context owns eligibility/budget.
// Heating manager remains the control algorithm owner.
FOR L_i := 1 TO GVL_CONSTANTS.C_MAX_MANIFOLDS DO
    IF GVL_SYSTEM_COORDINATION.G_Block_Heating OR (NOT fbDecision.VO_Manifold_Enabled[L_i]) THEN
        GVL_STATE.G_Manifold_Pumps[L_i] := FALSE;
        GVL_STATE.G_Manifold_Valves[L_i] := 0.0;

        FOR L_j := 1 TO GVL_CONSTANTS.C_MAX_HEATING_CIRCUITS DO
            IF GVL_CONFIG.G_HMI_FloorHeating_Configs[L_j].manifold_id = L_i THEN
                L_Zone_Valves[L_j] := FALSE;
            END_IF;
        END_FOR;
    END_IF;
END_FOR;

fbDHWManager(
    VI_System_Time_MS := GVL_STATUS.G_System_Time_MS,
    VI_Current_TOD := GVL_STATUS.G_Current_TOD,
    VI_IsActivePLC := GVL_STATUS.G_Is_Active_PLC,
    VI_Temp := GVL_STATE.G_DHW_Temp,
    VI_Pressure := GVL_STATE.G_DHW_Pressure,
    VI_Config := GVL_CONFIG.G_DHW_Config,
    VI_Current_Day_Of_Week := GVL_STATUS.G_Current_Day,
    VI_IO_Modules_Online := GVL_STATUS.G_IO_Modules_Online,
    VI_Reset_Errors := GVL_INTENT_USER.I_Reset_Errors,
    VI_Emergency_Stop := GVL_STATE.G_Safety_Emergency_Stop,
    VI_System_Mode := GVL_STATE.G_System_Mode,
    VO_Heating_Pump => GVL_STATE.G_DHW_Heating_Pump,
    VO_Circ_Pump => GVL_STATE.G_DHW_Circ_Pump,
    VO_Status => GVL_STATUS.G_DHW_Status
);

// ============================================================
// S3. DIAGNOSTICS PROJECTION + EVENTS
// ============================================================

GVL_STATUS.G_Diagnostics.Backup_Pump_Out_Of_Service := NOT GVL_CONFIG.G_Backup_Circulation_Pump_In_Service;
GVL_STATUS.G_Diagnostics.Electric_Heater_Out_Of_Service := NOT GVL_CONFIG.G_Electric_Heater_In_Service;

fbDiagEventManager(
    VI_Code := GVL_CONFIG.ERR_BACKUP_PUMP_OUT_OF_SERVICE,
    VI_Severity := 2,
    VI_Active := NOT GVL_CONFIG.G_Backup_Circulation_Pump_In_Service,
    VI_Timestamp := GVL_STATUS.G_System_Time_MS,
    VI_Source := 400,
    VIO_Events := GVL_STATUS.G_Diagnostics_Events,
    VIO_Count := GVL_STATUS.G_Diagnostics_Count
);

fbDiagEventManager(
    VI_Code := GVL_CONFIG.ERR_ELECTRIC_HEATER_OUT_OF_SERVICE,
    VI_Severity := 2,
    VI_Active := NOT GVL_CONFIG.G_Electric_Heater_In_Service,
    VI_Timestamp := GVL_STATUS.G_System_Time_MS,
    VI_Source := 401,
    VIO_Events := GVL_STATUS.G_Diagnostics_Events,
    VIO_Count := GVL_STATUS.G_Diagnostics_Count
);

FOR L_i := 1 TO GVL_CONSTANTS.C_MAX_MANIFOLDS DO
    GVL_STATUS.G_Diagnostics.Manifold_Pump_Out_Of_Service[L_i] := NOT GVL_CONFIG.G_Manifold_Pump_In_Service[L_i];

    fbDiagEventManager(
        VI_Code := GVL_CONFIG.ERR_MANIFOLD_PUMP_OUT_OF_SERVICE,
        VI_Severity := 2,
        VI_Active := NOT GVL_CONFIG.G_Manifold_Pump_In_Service[L_i],
        VI_Timestamp := GVL_STATUS.G_System_Time_MS,
        VI_Source := 410 + L_i,
        VIO_Events := GVL_STATUS.G_Diagnostics_Events,
        VIO_Count := GVL_STATUS.G_Diagnostics_Count
    );
END_FOR;

GVL_STATUS.G_Diagnostics.DHW_Heating_Pump_Out_Of_Service := NOT GVL_CONFIG.G_DHW_Heating_Pump_In_Service;
GVL_STATUS.G_Diagnostics.DHW_Circ_Pump_Out_Of_Service := NOT GVL_CONFIG.G_DHW_Circ_Pump_In_Service;

fbDiagEventManager(
    VI_Code := GVL_CONFIG.ERR_DHW_HEATING_PUMP_OUT_OF_SERVICE,
    VI_Severity := 2,
    VI_Active := NOT GVL_CONFIG.G_DHW_Heating_Pump_In_Service,
    VI_Timestamp := GVL_STATUS.G_System_Time_MS,
    VI_Source := 420,
    VIO_Events := GVL_STATUS.G_Diagnostics_Events,
    VIO_Count := GVL_STATUS.G_Diagnostics_Count
);

fbDiagEventManager(
    VI_Code := GVL_CONFIG.ERR_DHW_CIRC_PUMP_OUT_OF_SERVICE,
    VI_Severity := 2,
    VI_Active := NOT GVL_CONFIG.G_DHW_Circ_Pump_In_Service,
    VI_Timestamp := GVL_STATUS.G_System_Time_MS,
    VI_Source := 421,
    VIO_Events := GVL_STATUS.G_Diagnostics_Events,
    VIO_Count := GVL_STATUS.G_Diagnostics_Count
);

fbDiagEventManager(
    VI_Code := GVL_CONFIG.ERR_FREEZE_HARDWARE_FAILED,
    VI_Severity := 4,
    VI_Active := GVL_STATE.G_Freeze_Hardware_Failed,
    VI_Timestamp := GVL_STATUS.G_System_Time_MS,
    VI_Source := 430,
    VIO_Events := GVL_STATUS.G_Diagnostics_Events,
    VIO_Count := GVL_STATUS.G_Diagnostics_Count
);

// ============================================================
// S4. MAINTENANCE GATING
// ============================================================

IF NOT GVL_CONFIG.G_Backup_Circulation_Pump_In_Service THEN
    GVL_STATE.G_Backup_Circulation_Pump := FALSE;
END_IF;
IF NOT GVL_CONFIG.G_Electric_Heater_In_Service THEN
    GVL_STATE.G_Electric_Heater_Enable := FALSE;
END_IF;
FOR L_i := 1 TO GVL_CONSTANTS.C_MAX_MANIFOLDS DO
    IF NOT GVL_CONFIG.G_Manifold_Pump_In_Service[L_i] THEN
        GVL_STATE.G_Manifold_Pumps[L_i] := FALSE;
    END_IF;
END_FOR;
IF NOT GVL_CONFIG.G_DHW_Heating_Pump_In_Service THEN
    GVL_STATE.G_DHW_Heating_Pump := FALSE;
END_IF;
IF NOT GVL_CONFIG.G_DHW_Circ_Pump_In_Service THEN
    GVL_STATE.G_DHW_Circ_Pump := FALSE;
END_IF;

// ============================================================
// S5. FREEZE HARDWARE SUPPORT LOGIC
// ============================================================

GVL_STATE.G_Freeze_Hardware_Degraded := GVL_STATUS.G_Diagnostics.Backup_Pump_Fault OR GVL_STATUS.G_Diagnostics.Electric_Heater_Fault;
GVL_STATE.G_Freeze_Hardware_Failed := GVL_STATUS.G_Diagnostics.Backup_Pump_Fault AND GVL_STATUS.G_Diagnostics.Electric_Heater_Fault;
IF GVL_STATE.G_Freeze_Hardware_Failed THEN
    GVL_STATE.G_Backup_Circulation_Pump := FALSE;
    GVL_STATE.G_Electric_Heater_Enable := FALSE;
    GVL_STATE.G_Safety_Freeze_Risk := TRUE;
END_IF;

// >>> BULK_SYNC_ANCHOR: PRG_Heating <<<

// ============================================================
// S6. ADAPTER COPY-OUT
// ============================================================

FOR L_i := 1 TO GVL_CONSTANTS.C_MAX_HEATING_CIRCUITS DO
    GVL_STATE.G_Zone_Valves[L_i] := L_Zone_Valves[L_i];
END_FOR;
          
END_PROGRAM

PROGRAM PRG_Safety
  VAR
    fbWaterLeakageManager : FB_Water_Leakage_Manager;
    fbGasSmokeManager : FB_Gas_Smoke_Manager;
    fbSafetyWorkflow : FB_Safety_Workflow_Manager;
    fbOwnership : FB_Ownership_Watchdog;
    L_i : INT;
  END_VAR

            // ========================================
// SAFETY_INTENT_RESET_INIT
// ========================================
GVL_INTENT_SAFETY.I_Source_Valid := TRUE;
GVL_INTENT_SAFETY.I_Last_Update_MS := GVL_STATUS.G_System_Time_MS;
GVL_INTENT_SAFETY.I_Fire_Alarm_Active := FALSE;
GVL_INTENT_SAFETY.I_Gas_Alarm_Active := FALSE;
GVL_INTENT_SAFETY.I_Leak_Alarm_Active := FALSE;
GVL_INTENT_SAFETY.I_CO_Warning_Active := FALSE;
GVL_INTENT_SAFETY.I_System_Safe_Stop_Required := FALSE;
GVL_INTENT_SAFETY.I_Freeze_Protection_Required := FALSE;
GVL_INTENT_SAFETY.I_Evacuation_Mode_Active := FALSE;
GVL_INTENT_SAFETY.I_Gas_Close_Required := FALSE;
GVL_INTENT_SAFETY.I_Boiler_Stop_Required := FALSE;
GVL_INTENT_SAFETY.I_Vent_Stop_Required := FALSE;
GVL_INTENT_SAFETY.I_Vent_Force_PV3_Boost := FALSE;
GVL_INTENT_SAFETY.I_Vent_Force_Supply_100 := FALSE;
GVL_INTENT_SAFETY.I_Vent_Force_Supply_80 := FALSE;
GVL_INTENT_SAFETY.I_Vent_Force_Exhaust_100 := FALSE;
GVL_INTENT_SAFETY.I_Water_Main_Close_Required := FALSE;
GVL_INTENT_SAFETY.I_Water_Selective_Recovery_Allowed := FALSE;
GVL_INTENT_SAFETY.I_Water_Recovery_Target_Zone := 0;
GVL_INTENT_SAFETY.I_Lock_1_Force_Open := FALSE;
GVL_INTENT_SAFETY.I_Lock_1_Force_Close_Block := FALSE;
GVL_INTENT_SAFETY.I_Lock_2_Force_Open := FALSE;
GVL_INTENT_SAFETY.I_Lock_2_Force_Close_Block := FALSE;

// ========================================
// SAFETY_WORKFLOW_FB
// ========================================
fbSafetyWorkflow(
    VI_System_Time_MS := GVL_STATUS.G_System_Time_MS,
    VI_Water_Selective_Recover := GVL_INTENT_USER.I_Water_Selective_Recover,
    VI_Gas_Selective_Recover := GVL_INTENT_USER.I_Gas_Selective_Recover,
    VI_Water_Valve_Test_Open := GVL_INTENT_USER.I_Water_Valve_Test_Open,
    VI_Water_Valve_Test_Close := GVL_INTENT_USER.I_Water_Valve_Test_Close,
    VI_Water_Valve_Test_Confirm := GVL_INTENT_USER.I_Water_Valve_Test_Confirm,
    VI_Gas_Valve_Test_Open := GVL_INTENT_USER.I_Gas_Valve_Test_Open,
    VI_Gas_Valve_Test_Close := GVL_INTENT_USER.I_Gas_Valve_Test_Close,
    VI_Gas_Valve_Test_Confirm := GVL_INTENT_USER.I_Gas_Valve_Test_Confirm
);

IF fbSafetyWorkflow.VO_Water_Test_Timeout_Close_Required THEN
    GVL_INTENT_SAFETY.I_Water_Main_Close_Required := TRUE;
END_IF;

IF fbSafetyWorkflow.VO_Gas_Test_Timeout_Close_Required THEN
    GVL_INTENT_SAFETY.I_Gas_Close_Required := TRUE;
END_IF;

// ========================================
// SAFETY_DETECTORS_AND_HEALTH_PROJECTION
// ========================================
fbWaterLeakageManager(
    VI_System_Time_MS := GVL_STATUS.G_System_Time_MS,
    VI_IsActivePLC := GVL_STATUS.G_Is_Active_PLC,
    VI_Sensors := GVL_STATE.G_Water_Sensors,
    VI_Config := GVL_CONFIG.G_HMI_Flood_Config,
    VO_Status_Msg => GVL_STATUS.G_Flood_Status_Msg,
    VO_Leak_Detected => GVL_HEALTH_BRIDGE.G_Leak_Detected,
    VO_Leak_Warning_Level => GVL_HEALTH_BRIDGE.G_Leak_Warning_Level
);
GVL_INTENT_SAFETY.I_Leak_Alarm_Active := GVL_HEALTH_BRIDGE.G_Leak_Detected;

fbGasSmokeManager(
    VI_System_Time_MS := GVL_STATUS.G_System_Time_MS,
    VI_IsActivePLC := GVL_STATUS.G_Is_Active_PLC,
    VI_Methane_LEL := GVL_Safety_Selector.G_Methane_Effective_Array,
    VI_CO_PPM := GVL_Safety_Selector.G_CO_Effective_Array,
    VI_Smoke_Sensors := GVL_Safety_Selector.G_Smoke_Effective_Array,
    VI_Mute_Request := GVL_CONFIG.G_HMI_Mute_Alarm,
    VO_Smoke_Detected => GVL_HEALTH_BRIDGE.G_Smoke_Detected,
    VO_Gas_Detected => GVL_HEALTH_BRIDGE.G_Gas_Detected,
    VO_CO_Warning_Level => GVL_HEALTH_BRIDGE.G_CO_Warning_Level,
    VO_CO_Alarm_Level => GVL_HEALTH_BRIDGE.G_CO_Alarm_Level,
    VO_Status_Msg => GVL_STATUS.G_Gas_Status_Msg
);
GVL_INTENT_SAFETY.I_Fire_Alarm_Active := GVL_HEALTH_BRIDGE.G_Smoke_Detected;
GVL_INTENT_SAFETY.I_Gas_Alarm_Active := GVL_HEALTH_BRIDGE.G_Gas_Detected OR GVL_HEALTH_BRIDGE.G_CO_Alarm_Level;
GVL_INTENT_SAFETY.I_CO_Warning_Active := GVL_HEALTH_BRIDGE.G_CO_Warning_Level;

// ========================================
// OWNERSHIP WATCHDOG
// ========================================
fbOwnership(
    VI_Gas_Level := GVL_STATE.G_Methane_Sensors[1],
    VI_Gas_Alarm := GVL_STATE.G_Safety_Gas_Alarm,
    VI_Leak_Alarm := GVL_STATE.G_Safety_Leak_Alarm,
    VI_Smoke_Alarm := GVL_STATE.G_Safety_Smoke_Alarm
);

IF fbOwnership.VO_Ownership_Violation THEN
    GVL_TEST.G_Ownership_Violation := TRUE;
END_IF;

// ========================================
// SAFETY_CORE_HAZARD_INTERLOCK_PROJECTION
// ========================================
IF GVL_STATE.G_Safety_Smoke_Latched THEN
    GVL_INTENT_SAFETY.I_System_Safe_Stop_Required := TRUE;
    GVL_INTENT_SAFETY.I_Evacuation_Mode_Active := TRUE;
    GVL_INTENT_SAFETY.I_Boiler_Stop_Required := TRUE;
    GVL_INTENT_SAFETY.I_Vent_Stop_Required := TRUE;
    GVL_INTENT_SAFETY.I_Lock_1_Force_Open := TRUE;
    GVL_INTENT_SAFETY.I_Lock_1_Force_Close_Block := TRUE;
    GVL_INTENT_SAFETY.I_Lock_2_Force_Open := TRUE;
    GVL_INTENT_SAFETY.I_Lock_2_Force_Close_Block := TRUE;
END_IF;

IF GVL_STATE.G_Safety_Gas_Latched THEN
    GVL_INTENT_SAFETY.I_System_Safe_Stop_Required := TRUE;
    GVL_INTENT_SAFETY.I_Gas_Close_Required := TRUE;
    GVL_INTENT_SAFETY.I_Boiler_Stop_Required := TRUE;
    GVL_INTENT_SAFETY.I_Vent_Force_PV3_Boost := TRUE;
    GVL_INTENT_SAFETY.I_Vent_Force_Supply_100 := TRUE;
END_IF;

IF GVL_HEALTH_BRIDGE.G_CO_Warning_Level OR GVL_HEALTH_BRIDGE.G_CO_Alarm_Level THEN
    GVL_INTENT_SAFETY.I_Vent_Force_Supply_80 := TRUE;
END_IF;

IF GVL_STATE.G_Safety_Leak_Latched THEN
    GVL_INTENT_SAFETY.I_Water_Main_Close_Required := TRUE;
END_IF;

// ========================================
// SAFETY_RESIDUAL_NON_WORKFLOW_PROJECTION
// ========================================
IF GVL_STATE.G_Freeze_Hardware_Degraded THEN
    GVL_INTENT_SAFETY.I_Freeze_Protection_Required := TRUE;
END_IF;

// >>> BULK_SYNC_ANCHOR: PRG_Safety <<<
          
END_PROGRAM

PROGRAM PRG_Test_Injection

            // Non-intrusive test injection layer
// Must be called AFTER PRG_IO_Read and BEFORE PRG_Safety

IF NOT GVL_TEST_INJECTION.G_Inject_Enable THEN
    RETURN;
END_IF;

// ===== GAS INJECTION =====
IF GVL_TEST_INJECTION.G_Inject_Gas_Level > 0.0 THEN
    GVL_STATE.G_Methane_Sensors[1] := GVL_TEST_INJECTION.G_Inject_Gas_Level;
END_IF;

// ===== IO OFFLINE INJECTION =====
IF GVL_TEST_INJECTION.G_Inject_Force_IO_Offline THEN
    GVL_STATUS.G_IO_Modules_Online[1] := FALSE;
    GVL_STATUS.G_IO_Modules_Online[2] := FALSE;
END_IF;

// ===== OWNERSHIP VIOLATION TEST =====
// Intentionally break safety to verify watchdog
IF GVL_TEST_INJECTION.G_Inject_Force_Gas_Alarm_Reset THEN
    GVL_STATE.G_Safety_Gas_Alarm := FALSE;
END_IF;
          
END_PROGRAM

PROGRAM PRG_IO_Read
  VAR
    L_i : INT;
    L_Debounce_Time : TIME := T#100MS;
    L_Manifold_Pressure_Raw : WORD;
    L_Manifold_Current_Raw : WORD;
    fbDebounce_Switches : ARRAY[1..8] OF FB_System_Timer;
    fbDebounce_Motion : ARRAY[1..8] OF FB_System_Timer;
    fbDebounce_Security_Open : ARRAY[1..GVL_CONSTANTS.C_MAX_SECURITY_SENSORS] OF FB_System_Timer;
    fbDebounce_Security_Glass : ARRAY[1..GVL_CONSTANTS.C_MAX_SECURITY_SENSORS] OF FB_System_Timer;
    fbDebounce_Flood : ARRAY[1..GVL_CONSTANTS.C_MAX_FLOOD_SENSORS] OF FB_System_Timer;
    fbDebounce_Smoke : ARRAY[1..GVL_CONSTANTS.C_MAX_SMOKE_SENSORS] OF FB_System_Timer;
    fbDebounce_Group_2F : FB_System_Timer;
    fbIO_Watchdog_1 : FB_IO_Module_Watchdog;
    fbIO_Watchdog_2 : FB_IO_Module_Watchdog;
    fbDiagEventManager : FB_Diagnostics_Event_Manager;
    L_IO_Error_Active : BOOL;
    fbCalib_Outdoor_Temp : FB_Sensor_Calibration_Processor;
    fbCalib_Supply_Temps : ARRAY[1..GVL_CONSTANTS.C_MAX_SUPPLY_TEMPS] OF FB_Sensor_Calibration_Processor;
    fbCalib_Room_Temps : ARRAY[1..GVL_CONSTANTS.C_MAX_ZONES] OF FB_Sensor_Calibration_Processor;
    fbCalib_Floor_Temps : ARRAY[1..GVL_CONSTANTS.C_MAX_ZONES] OF FB_Sensor_Calibration_Processor;
    fbCalib_Room_Hum : ARRAY[1..GVL_CONSTANTS.C_MAX_ZONES] OF FB_Sensor_Calibration_Processor;
    fbCalib_Room_CO2 : ARRAY[1..GVL_CONSTANTS.C_MAX_ZONES] OF FB_Sensor_Calibration_Processor;
    fbCalib_Manifold_T_Supply : ARRAY[1..GVL_CONSTANTS.C_MAX_MANIFOLDS] OF FB_Sensor_Calibration_Processor;
    fbCalib_Manifold_T_Return : ARRAY[1..GVL_CONSTANTS.C_MAX_MANIFOLDS] OF FB_Sensor_Calibration_Processor;
    fbCalib_Methane : ARRAY[1..GVL_CONSTANTS.C_MAX_METHANE_SENSORS] OF FB_Sensor_Calibration_Processor;
    fbCalib_CO : ARRAY[1..GVL_CONSTANTS.C_MAX_CO_SENSORS] OF FB_Sensor_Calibration_Processor;
    fbAnalog_Manifold_Pressure : ARRAY[1..GVL_CONSTANTS.C_MAX_MANIFOLDS] OF FB_Sensor_Analog_Processing;
    fbAnalog_Manifold_Current : ARRAY[1..GVL_CONSTANTS.C_MAX_MANIFOLDS] OF FB_Sensor_Analog_Processing;
  END_VAR

            // ===== ORIGINAL SNAPSHOT (FULL) =====
fbIO_Watchdog_1(VI_System_Time_MS := GVL_STATUS.G_System_Time_MS, VI_Module_ID := 1, VI_Heartbeat_Signal := GVL_IO.DI_Module_1_Heartbeat, VI_Timeout_MS := 2000);
fbIO_Watchdog_2(VI_System_Time_MS := GVL_STATUS.G_System_Time_MS, VI_Module_ID := 2, VI_Heartbeat_Signal := GVL_IO.DI_Module_2_Heartbeat, VI_Timeout_MS := 2000);

GVL_STATUS.G_IO_Modules_Online[1] := fbIO_Watchdog_1.VO_Module_Online;
GVL_STATUS.G_IO_Modules_Online[2] := fbIO_Watchdog_2.VO_Module_Online;

L_IO_Error_Active := fbIO_Watchdog_1.VO_Error_Active OR fbIO_Watchdog_2.VO_Error_Active;

// IO watchdog events
fbDiagEventManager(
    VI_Code := 16#E001,
    VI_Severity := 4,
    VI_Active := NOT fbIO_Watchdog_1.VO_Module_Online,
    VI_Timestamp := GVL_STATUS.G_System_Time_MS,
    VI_Source := 1,
    VIO_Events := GVL_STATUS.G_Diagnostics_Events,
    VIO_Count := GVL_STATUS.G_Diagnostics_Count
);

fbDiagEventManager(
    VI_Code := 16#E002,
    VI_Severity := 4,
    VI_Active := NOT fbIO_Watchdog_2.VO_Module_Online,
    VI_Timestamp := GVL_STATUS.G_System_Time_MS,
    VI_Source := 2,
    VIO_Events := GVL_STATUS.G_Diagnostics_Events,
    VIO_Count := GVL_STATUS.G_Diagnostics_Count
);

IF L_IO_Error_Active THEN
    GVL_COMMAND.G_Gas_Valve_Close := TRUE;
    GVL_COMMAND.G_Close_Valve_35 := TRUE;
    GVL_COMMAND.G_Close_Valve_36 := TRUE;
    FOR L_i := 1 TO GVL_CONSTANTS.C_MAX_MANIFOLDS DO GVL_STATE.G_Manifold_Pumps[L_i] := FALSE; END_FOR;
END_IF;

FOR L_i := 1 TO 8 DO
    fbDebounce_Switches[L_i](IN := GVL_IO.DI_Lighting_Switches[L_i], PT := L_Debounce_Time, VI_System_Time_MS := GVL_STATUS.G_System_Time_MS);
    GVL_STATE.G_Physical_Switches[L_i] := fbDebounce_Switches[L_i].Q;
    
    fbDebounce_Motion[L_i](IN := GVL_IO.DI_Motion_Sensors[L_i], PT := L_Debounce_Time, VI_System_Time_MS := GVL_STATUS.G_System_Time_MS);
    GVL_STATE.G_Motion_Sensors[L_i] := fbDebounce_Motion[L_i].Q;
END_FOR;

FOR L_i := 1 TO GVL_CONSTANTS.C_MAX_SOCKETS DO
    GVL_STATE.G_Socket_Switches[L_i] := FALSE;
END_FOR;

FOR L_i := 1 TO GVL_CONSTANTS.C_MAX_SECURITY_SENSORS DO
    fbDebounce_Security_Open[L_i](IN := GVL_IO.DI_Security_Open[L_i], PT := L_Debounce_Time, VI_System_Time_MS := GVL_STATUS.G_System_Time_MS);
    fbDebounce_Security_Glass[L_i](IN := GVL_IO.DI_Security_Glass[L_i], PT := L_Debounce_Time, VI_System_Time_MS := GVL_STATUS.G_System_Time_MS);
END_FOR;

fbDebounce_Group_2F(IN := GVL_IO.DI_Security_2F_Group, PT := L_Debounce_Time, VI_System_Time_MS := GVL_STATUS.G_System_Time_MS);

FOR L_i := 1 TO GVL_CONSTANTS.C_MAX_DOOR_SENSORS DO
    IF GVL_CONFIG.G_Door_Map[L_i] > 0 AND GVL_CONFIG.G_Door_Map[L_i] <= GVL_CONSTANTS.C_MAX_SECURITY_SENSORS THEN
        GVL_STATE.G_Door_Sensors[L_i] := fbDebounce_Security_Open[GVL_CONFIG.G_Door_Map[L_i]].Q;
    END_IF;
END_FOR;

FOR L_i := 1 TO 8 DO
    IF GVL_CONFIG.G_Window_Map[L_i] > 0 THEN
        IF GVL_CONFIG.G_Window_Map[L_i] <= GVL_CONSTANTS.C_MAX_SECURITY_SENSORS THEN
            GVL_STATE.G_Window_Sensors[L_i] := fbDebounce_Security_Open[GVL_CONFIG.G_Window_Map[L_i]].Q;
        ELSE
            GVL_STATE.G_Window_Sensors[L_i] := fbDebounce_Security_Glass[GVL_CONFIG.G_Window_Map[L_i] - GVL_CONSTANTS.C_MAX_SECURITY_SENSORS].Q;
        END_IF;
    END_IF;
END_FOR;
GVL_STATE.G_Window_Sensors[16] := fbDebounce_Group_2F.Q;

FOR L_i := 1 TO GVL_CONSTANTS.C_MAX_FLOOD_SENSORS DO
    fbDebounce_Flood[L_i](IN := GVL_IO.DI_Flood_Sensors[L_i], PT := L_Debounce_Time, VI_System_Time_MS := GVL_STATUS.G_System_Time_MS);
    GVL_STATE.G_Water_Sensors[L_i] := fbDebounce_Flood[L_i].Q;
END_FOR;

FOR L_i := 1 TO GVL_CONSTANTS.C_MAX_SMOKE_SENSORS DO
    fbDebounce_Smoke[L_i](IN := GVL_IO.DI_Smoke_Sensors[L_i], PT := L_Debounce_Time, VI_System_Time_MS := GVL_STATUS.G_System_Time_MS);
    GVL_STATE.G_Smoke_Sensors[L_i] := fbDebounce_Smoke[L_i].Q;
END_FOR;

// ===== ENHANCED LAYER =====
fbCalib_Outdoor_Temp(
    VI_Raw_Value := GVL_IO.AI_Temp_Outdoor.rValue,
    VI_Record := GVL_CONFIG.G_Calib_Outdoor_Temp
);
GVL_STATE.G_Outdoor_Temp := fbCalib_Outdoor_Temp.VO_Calibrated_Value;

FOR L_i := 1 TO GVL_CONSTANTS.C_MAX_SUPPLY_TEMPS DO
    IF GVL_IO.AI_Supply_Temps[L_i].wStatus = 0 THEN
        fbCalib_Supply_Temps[L_i](
            VI_Raw_Value := GVL_IO.AI_Supply_Temps[L_i].rValue,
            VI_Record := GVL_CONFIG.G_Calib_Supply_Temps[L_i]
        );
        GVL_STATE.G_Supply_Temps[L_i] := fbCalib_Supply_Temps[L_i].VO_Calibrated_Value;
    END_IF;
END_FOR;

FOR L_i := 1 TO 8 DO
    fbCalib_Room_Hum[L_i](
        VI_Raw_Value := GVL_IO.AI_Room_Hum[L_i],
        VI_Record := GVL_CONFIG.G_Calib_Humidity[L_i]
    );
    GVL_STATE.G_Room_Hum[L_i] := fbCalib_Room_Hum[L_i].VO_Calibrated_Value;

    fbCalib_Room_CO2[L_i](
        VI_Raw_Value := GVL_IO.AI_Room_CO2[L_i],
        VI_Record := GVL_CONFIG.G_Calib_CO2[L_i]
    );
    GVL_STATE.G_Room_CO2[L_i] := fbCalib_Room_CO2[L_i].VO_Calibrated_Value;
END_FOR;

FOR L_i := 1 TO 8 DO
    fbCalib_Room_Temps[L_i](
        VI_Raw_Value := GVL_IO.AI_Room_Temps[L_i],
        VI_Record := GVL_CONFIG.G_Calib_Room_Temps[L_i]
    );
    GVL_STATE.G_Room_Temps[L_i] := fbCalib_Room_Temps[L_i].VO_Calibrated_Value;

    fbCalib_Floor_Temps[L_i](
        VI_Raw_Value := GVL_IO.AI_Floor_Temps[L_i],
        VI_Record := GVL_CONFIG.G_Calib_Floor_Temps[L_i]
    );
    GVL_STATE.G_Floor_Temps[L_i] := fbCalib_Floor_Temps[L_i].VO_Calibrated_Value;
END_FOR;

GVL_STATUS.G_Diagnostics.Manifold_Pressure_Fault_Active := FALSE;
GVL_STATUS.G_Diagnostics.Manifold_Pressure_First_Fault_Index := 0;
GVL_STATUS.G_Diagnostics.Manifold_Current_Fault_Active := FALSE;
GVL_STATUS.G_Diagnostics.Manifold_Current_First_Fault_Index := 0;
GVL_STATUS.G_Diagnostics.Manifold_Pressure_Fault_Text := '';
GVL_STATUS.G_Diagnostics.Manifold_Current_Fault_Text := '';
GVL_STATUS.G_Diagnostics.Sensor_Fault := FALSE;
GVL_STATUS.G_Diagnostics.Subsystem_Degraded := FALSE;

FOR L_i := 1 TO GVL_CONSTANTS.C_MAX_MANIFOLDS DO
    IF GVL_IO.AI_Manifold_Pressures[L_i] < 0 THEN
        L_Manifold_Pressure_Raw := 0;
    ELSE
        L_Manifold_Pressure_Raw := INT_TO_WORD(GVL_IO.AI_Manifold_Pressures[L_i]);
    END_IF;

    IF GVL_IO.AI_Manifold_Currents[L_i] < 0 THEN
        L_Manifold_Current_Raw := 0;
    ELSE
        L_Manifold_Current_Raw := INT_TO_WORD(GVL_IO.AI_Manifold_Currents[L_i]);
    END_IF;

    fbAnalog_Manifold_Pressure[L_i](
        VI_Raw_Value := L_Manifold_Pressure_Raw,
        VI_Sensor_Type := 0,
        VI_Min_Scale := 0.0,
        VI_Max_Scale := 10.0,
        VI_Offset := 0.0,
        VI_Multiplier := 1.0,
        VI_Filter_Time_MS := GVL_CONSTANTS.C_MS_IN_SECOND,
        VI_System_Time_MS := GVL_STATUS.G_System_Time_MS,
        VI_Fallback_Mode := 0,
        VI_Default_Value := 0.0
    );
    GVL_STATE.G_Manifold_Pressures[L_i] := fbAnalog_Manifold_Pressure[L_i].VO_Value;
    GVL_STATUS.G_Diagnostics.Manifold_Pressure_Fault[L_i] := fbAnalog_Manifold_Pressure[L_i].VO_Error;
    GVL_STATUS.G_Diagnostics.Manifold_Pressure_Diag_Code[L_i] := fbAnalog_Manifold_Pressure[L_i].VO_Diag_Code;

    fbDiagEventManager(
        VI_Code := GVL_CONFIG.ERR_PRESSURE_OUT_OF_RANGE,
        VI_Severity := 3,
        VI_Active := fbAnalog_Manifold_Pressure[L_i].VO_Error,
        VI_Timestamp := GVL_STATUS.G_System_Time_MS,
        VI_Source := 100 + L_i,
        VIO_Events := GVL_STATUS.G_Diagnostics_Events,
        VIO_Count := GVL_STATUS.G_Diagnostics_Count
    );

    fbAnalog_Manifold_Current[L_i](
        VI_Raw_Value := L_Manifold_Current_Raw,
        VI_Sensor_Type := 0,
        VI_Min_Scale := 0.0,
        VI_Max_Scale := 16.0,
        VI_Offset := 0.0,
        VI_Multiplier := 1.0,
        VI_Filter_Time_MS := GVL_CONSTANTS.C_MS_IN_SECOND,
        VI_System_Time_MS := GVL_STATUS.G_System_Time_MS,
        VI_Fallback_Mode := 0,
        VI_Default_Value := 0.0
    );
    GVL_STATE.G_Manifold_Currents[L_i] := fbAnalog_Manifold_Current[L_i].VO_Value;
    GVL_STATUS.G_Diagnostics.Manifold_Current_Fault[L_i] := fbAnalog_Manifold_Current[L_i].VO_Error;
    GVL_STATUS.G_Diagnostics.Manifold_Current_Diag_Code[L_i] := fbAnalog_Manifold_Current[L_i].VO_Diag_Code;

    fbDiagEventManager(
        VI_Code := GVL_CONFIG.ERR_PUMP_UNDERCURRENT,
        VI_Severity := 3,
        VI_Active := fbAnalog_Manifold_Current[L_i].VO_Error,
        VI_Timestamp := GVL_STATUS.G_System_Time_MS,
        VI_Source := 200 + L_i,
        VIO_Events := GVL_STATUS.G_Diagnostics_Events,
        VIO_Count := GVL_STATUS.G_Diagnostics_Count
    );

    IF GVL_IO.AI_Manifold_Temps_Supply[L_i].wStatus = 0 THEN
        fbCalib_Manifold_T_Supply[L_i](
            VI_Raw_Value := GVL_IO.AI_Manifold_Temps_Supply[L_i].rValue,
            VI_Record := GVL_CONFIG.G_Calib_Manifold_T_Supply[L_i]
        );
        GVL_STATE.G_Manifold_T_Supply[L_i] := fbCalib_Manifold_T_Supply[L_i].VO_Calibrated_Value;
    END_IF;

    fbCalib_Manifold_T_Return[L_i](
        VI_Raw_Value := INT_TO_REAL(GVL_IO.AI_Manifold_Temps_Return[L_i]) / 10.0,
        VI_Record := GVL_CONFIG.G_Calib_Manifold_T_Return[L_i]
    );
    GVL_STATE.G_Manifold_T_Return[L_i] := fbCalib_Manifold_T_Return[L_i].VO_Calibrated_Value;
    GVL_STATE.G_Manifold_End_Switches[L_i] := GVL_IO.DI_Manifold_End_Switches[L_i];

    IF GVL_STATUS.G_Diagnostics.Manifold_Pressure_Fault[L_i] OR GVL_STATUS.G_Diagnostics.Manifold_Current_Fault[L_i] THEN
        GVL_STATUS.G_Diagnostics.Sensor_Fault := TRUE;
        GVL_STATUS.G_Diagnostics.Subsystem_Degraded := TRUE;
    END_IF;

    IF GVL_STATUS.G_Diagnostics.Manifold_Pressure_Fault[L_i] AND GVL_STATUS.G_Diagnostics.Manifold_Current_Fault[L_i] THEN
        GVL_STATUS.G_Diagnostics.Manifold_Pressure_Fault_Text := 'Correlated pressure/current fault detected';
        GVL_STATUS.G_Diagnostics.Manifold_Current_Fault_Text := 'Correlated pressure/current fault detected';
    ELSIF GVL_STATUS.G_Diagnostics.Manifold_Pressure_Fault[L_i] AND (GVL_STATUS.G_Diagnostics.Manifold_Pressure_Fault_Text = '') THEN
        GVL_STATUS.G_Diagnostics.Manifold_Pressure_Fault_Text := 'Pressure sensor fault detected';
    ELSIF GVL_STATUS.G_Diagnostics.Manifold_Current_Fault[L_i] AND (GVL_STATUS.G_Diagnostics.Manifold_Current_Fault_Text = '') THEN
        GVL_STATUS.G_Diagnostics.Manifold_Current_Fault_Text := 'Current sensor fault detected';
    END_IF;
END_FOR;

FOR L_i := 1 TO GVL_CONSTANTS.C_MAX_METHANE_SENSORS DO
    IF GVL_IO.AI_Methane_LEL[L_i].wStatus = 0 THEN
        fbCalib_Methane[L_i](
            VI_Raw_Value := GVL_IO.AI_Methane_LEL[L_i].rValue,
            VI_Record := GVL_CONFIG.G_Calib_Methane[L_i]
        );
        GVL_STATE.G_Methane_Sensors[L_i] := fbCalib_Methane[L_i].VO_Calibrated_Value;
    END_IF;

    fbDiagEventManager(
        VI_Code := 16#E003,
        VI_Severity := 3,
        VI_Active := GVL_IO.AI_Methane_LEL[L_i].wStatus <> 0,
        VI_Timestamp := GVL_STATUS.G_System_Time_MS,
        VI_Source := 300 + L_i,
        VIO_Events := GVL_STATUS.G_Diagnostics_Events,
        VIO_Count := GVL_STATUS.G_Diagnostics_Count
    );
END_FOR;

FOR L_i := 1 TO GVL_CONSTANTS.C_MAX_CO_SENSORS DO
    fbCalib_CO[L_i](
        VI_Raw_Value := GVL_IO.AI_CO_PPM[L_i],
        VI_Record := GVL_CONFIG.G_Calib_CO[L_i]
    );
    GVL_STATE.G_CO_Sensors[L_i] := fbCalib_CO[L_i].VO_Calibrated_Value;
END_FOR;

GVL_STATE.G_Boiler_Flame := GVL_IO.AI_Boiler_Flame_Status;
GVL_STATE.G_Boiler_Error := GVL_IO.DI_Boiler_Error;
FOR L_i := 1 TO GVL_CONSTANTS.C_MAX_BOILERS DO
    GVL_STATE.G_Boiler_OT_Online[L_i] := FALSE;
END_FOR;

GVL_STATE.G_DHW_Temp := GVL_IO.AI_DHW_Temp;
GVL_STATE.G_DHW_Pressure := GVL_IO.AI_DHW_Pressure;

GVL_STATE.G_Water_Zone_Open_FB := GVL_IO.DI_Water_Zone_Open_FB;
GVL_STATE.G_Water_Zone_Close_FB := GVL_IO.DI_Water_Zone_Close_FB;

// >>> BULK_SYNC_ANCHOR: PRG_IO_Read <<<
          
END_PROGRAM

PROGRAM PRG_Security
  VAR
    L_i : INT;
    L_Motion_Sensors_16 : ARRAY[1..16] OF BOOL;
    fbSecurityManager : FB_Security_System_Manager;
    fbAccessControl : FB_Access_Control;
  END_VAR

            FOR L_i := 1 TO 16 DO
    L_Motion_Sensors_16[L_i] := GVL_STATE.G_Motion_Sensors[L_i];
END_FOR;
// 7. Система безопасности (Охранная сигнализация)
fbSecurityManager(
    VI_System_Time_MS := GVL_STATUS.G_System_Time_MS,
    VI_IsActivePLC := GVL_STATUS.G_Is_Active_PLC,
    VI_Motion_Sensors := L_Motion_Sensors_16,
    VI_Door_Sensors := GVL_STATE.G_Door_Sensors,
    VI_Window_Sensors := GVL_STATE.G_Window_Sensors,
    VI_Arm_Request := GVL_INTENT_USER.I_Arm_Request,
    VI_Disarm_Request := GVL_INTENT_USER.I_Disarm_Request,
    VI_PIN_Code := GVL_INTENT_USER.I_PIN_Code,
    VI_RFID_Tag := GVL_INTENT_USER.I_RFID_Tag,
    VI_2FA_Code := GVL_INTENT_USER.I_2FA_Code_In,
    VI_Config := GVL_CONFIG.G_Security_Config,
    VI_Bypass_Motion := GVL_CONFIG.G_Security_Config.bypass_motion,
    VI_Bypass_Doors := GVL_CONFIG.G_Security_Config.bypass_doors,
    VI_Bypass_Windows := GVL_CONFIG.G_Security_Config.bypass_windows,
    VI_Current_TOD := GVL_STATUS.G_Current_TOD,
    VO_Armed => GVL_ALARM.G_Security_Armed,
    VO_Alarm_Active => GVL_ALARM.G_Security_Alarm,
    VO_Siren_Active => GVL_ALARM.G_Security_Siren,
    VO_Status_Msg => GVL_STATUS.G_Security_Status_Msg,
    VO_Send_Code_Req => GVL_COMMAND.G_Send_2FA_Req,
    VO_Code_To_Send => GVL_COMMAND.G_2FA_Code_Out
);

// 7.1 Контроль доступа (СКУД)
fbAccessControl(
    VI_System_Time_MS := GVL_STATUS.G_System_Time_MS,
    VI_IsActivePLC := GVL_STATUS.G_Is_Active_PLC,
    VI_Armed := GVL_ALARM.G_Security_Armed,
    VI_System_Mode := GVL_STATE.G_System_Mode,
    VI_Gate_Open_Req := GVL_CONFIG.G_HMI_Gate_Open_Req,
    VI_Wicket_Open_Req := GVL_CONFIG.G_HMI_Wicket_Open_Req,
    VI_Lock_1_Open_Req := GVL_CONFIG.G_HMI_Lock_1_Open_Req,
    VI_Lock_1_Close_Req := GVL_CONFIG.G_HMI_Lock_1_Close_Req,
    VI_Lock_2_Open_Req := GVL_CONFIG.G_HMI_Lock_2_Open_Req,
    VI_Lock_2_Close_Req := GVL_CONFIG.G_HMI_Lock_2_Close_Req,
    VI_PIN_Code := GVL_INTENT_USER.I_PIN_Code,
    VI_RFID_Tag := GVL_INTENT_USER.I_RFID_Tag,
    VI_Access_Codes := GVL_Retain.G_Access_Codes,
    VI_RFID_Tags := GVL_Retain.G_RFID_Tags,
    VI_Config := GVL_CONFIG.G_Security_Config,
    VO_Gate_Open => GVL_INTENT_USER.I_Gate_Open_Request,
    VO_Wicket_Open => GVL_INTENT_USER.I_Wicket_Open_Request,
    VO_Lock_1_Open => GVL_INTENT_USER.I_Lock_1_Open_Request,
    VO_Lock_1_Close => GVL_INTENT_USER.I_Lock_1_Close_Request,
    VO_Lock_2_Open => GVL_INTENT_USER.I_Lock_2_Open_Request,
    VO_Lock_2_Close => GVL_INTENT_USER.I_Lock_2_Close_Request
);
          
END_PROGRAM

PROGRAM PRG_Presence_Manager
  VAR
    fbPresence : FB_Presence_Manager;
    L_i : INT;
  END_VAR

            fbPresence(
    VI_Motion_Sensors := GVL_STATE.G_Motion_Sensors,
    VI_System_Time_MS := GVL_STATUS.G_System_Time_MS
);

GVL_PRESENCE.G_Any_Motion := fbPresence.VO_Any_Motion;
GVL_PRESENCE.G_Occupied := fbPresence.VO_Occupied;
GVL_PRESENCE.G_Auto_Away_Request := fbPresence.VO_Auto_Away;
GVL_PRESENCE.G_Last_Motion_TS := fbPresence.VO_Last_Motion_TS;

FOR L_i := 1 TO GVL_CONSTANTS.C_MAX_ZONES DO
    IF GVL_STATE.G_Motion_Sensors[L_i] THEN
        GVL_PRESENCE.G_Zone_Occupied[L_i] := TRUE;
        GVL_PRESENCE.G_Zone_Last_Motion_TS[L_i] := GVL_STATUS.G_System_Time_MS;
    END_IF;

    IF (GVL_STATUS.G_System_Time_MS - GVL_PRESENCE.G_Zone_Last_Motion_TS[L_i]) > 900000 THEN
        GVL_PRESENCE.G_Zone_Occupied[L_i] := FALSE;
    END_IF;
END_FOR;
          
END_PROGRAM

PROGRAM PRG_Command_Arbitration
  VAR
    L_i : INT;
  END_VAR

            // Reset shadow operational commands before each arbitration cycle
GVL_COMMAND_SHADOW.G_Gas_Valve_Close := FALSE;
GVL_COMMAND_SHADOW.G_Boiler_Stop := FALSE;
GVL_COMMAND_SHADOW.G_Supply_100_Req := FALSE;
GVL_COMMAND_SHADOW.G_Supply_80_Req := FALSE;
GVL_COMMAND_SHADOW.G_Vent_PV3_Boost := FALSE;
GVL_COMMAND_SHADOW.G_Exhaust_100_Req := FALSE;
GVL_COMMAND_SHADOW.G_Vent_Stop := FALSE;

GVL_COMMAND_SHADOW.G_Close_Valve_35 := FALSE;
GVL_COMMAND_SHADOW.G_Close_Valve_36 := FALSE;

GVL_COMMAND_SHADOW.G_Lock_1_Open := FALSE;
GVL_COMMAND_SHADOW.G_Lock_1_Close := FALSE;
GVL_COMMAND_SHADOW.G_Lock_2_Open := FALSE;
GVL_COMMAND_SHADOW.G_Lock_2_Close := FALSE;
GVL_COMMAND_SHADOW.G_Gate_Open := FALSE;
GVL_COMMAND_SHADOW.G_Wicket_Open := FALSE;

